  MoveL 10150 to (-40.71, 50.09, 144.49) mm, rotated rx 180 ry 0 rz 180 deg; joints [-39.518, -30.421, 107.234, 74.541, 41.316, -69.786]
  MoveL 10151 to (-40.71, 50.09, 144.49) mm, rotated rx 180 ry 0 rz 180 deg; joints [-39.518, -30.421, 107.234, 74.541, 41.316, -69.786]
  Call Extruder(450.78136)
  MoveL 10152 to (-40.66, 49.79, 144.49) mm, rotated rx -180 ry 0 rz 180 deg; joints [-39.46, -30.443, 107.245, 74.499, 41.265, -69.747]
  MoveL 10153 to (-40.66, 49.79, 144.49) mm, rotated rx -180 ry 0 rz 180 deg; joints [-39.46, -30.443, 107.245, 74.499, 41.265, -69.747]
  Call Extruder(450.94309)
  MoveL 10154 to (-40.61, 49.48, 144.49) mm, rotated rx 180 ry 0 rz 180 deg; joints [-39.402, -30.465, 107.257, 74.456, 41.213, -69.708]
  MoveL 10155 to (-40.61, 49.48, 144.49) mm, rotated rx 180 ry 0 rz 180 deg; joints [-39.402, -30.465, 107.257, 74.456, 41.213, -69.708]
  Call Extruder(451.10554)
  MoveL 10156 to (-40.56, 49.18, 144.49) mm, rotated rx 180 ry 0 rz 180 deg; joints [-39.344, -30.487, 107.268, 74.413, 41.162, -69.669]
  MoveL 10157 to (-40.56, 49.18, 144.49) mm, rotated rx 180 ry 0 rz 180 deg; joints [-39.344, -30.487, 107.268, 74.413, 41.162, -69.669]
  Call Extruder(451.23946)
  MoveL 10158 to (-40.52, 48.93, 144.49) mm, rotated rx 180 ry 0 rz 180 deg; joints [-39.296, -30.504, 107.276, 74.378, 41.118, -69.637]
  MoveL 10159 to (-40.52, 48.93, 144.49) mm, rotated rx 180 ry 0 rz 180 deg; joints [-39.296, -30.504, 107.276, 74.378, 41.118, -69.637]
  Call Extruder(451.37400)
  MoveL 10160 to (-40.47, 48.68, 144.49) mm, rotated rx -180 ry 0 rz 180 deg; joints [-39.247, -30.521, 107.285, 74.343, 41.075, -69.605]
  MoveL 10161 to (-40.47, 48.68, 144.49) mm, rotated rx -180 ry 0 rz 180 deg; joints [-39.247, -30.521, 107.285, 74.343, 41.075, -69.605]
  Call Extruder(451.50914)
  MoveL 10162 to (-40.42, 48.43, 144.49) mm, rotated rx 180 ry 0 rz 180 deg; joints [-39.198, -30.538, 107.293, 74.308, 41.031, -69.574]
  MoveL 10163 to (-40.42, 48.43, 144.49) mm, rotated rx 180 ry 0 rz 180 deg; joints [-39.198, -30.538, 107.293, 74.308, 41.031, -69.574]
  Call Extruder(451.64490)
  MoveL 10164 to (-40.37, 48.18, 144.49) mm, rotated rx 180 ry 0 rz 180 deg; joints [-39.149, -30.555, 107.302, 74.273, 40.988, -69.542]
  MoveL 10165 to (-40.37, 48.18, 144.49) mm, rotated rx 180 ry 0 rz 180 deg; joints [-39.149, -30.555, 107.302, 74.273, 40.988, -69.542]
  Call Extruder(451.78127)
  MoveL 10166 to (-40.32, 47.93, 144.49) mm, rotated rx 180 ry 0 rz 180 deg; joints [-39.1, -30.572, 107.31, 74.237, 40.944, -69.51]
  MoveL 10167 to (-40.32, 47.93, 144.49) mm, rotated rx 180 ry 0 rz 180 deg; joints [-39.1, -30.572, 107.31, 74.237, 40.944, -69.51]
  Call Extruder(451.91824)
  MoveL 10168 to (-40.27, 47.68, 144.49) mm, rotated rx 180 ry 0 rz 180 deg; joints [-39.051, -30.589, 107.319, 74.202, 40.901, -69.478]
  MoveL 10169 to (-40.27, 47.68, 144.49) mm, rotated rx 180 ry 0 rz 180 deg; joints [-39.051, -30.589, 107.319, 74.202, 40.901, -69.478]
  Call Extruder(452.05583)
  MoveL 10170 to (-40.22, 47.43, 144.49) mm, rotated rx -180 ry 0 rz -180 deg; joints [-39.002, -30.605, 107.327, 74.166, 40.857, -69.446]
  MoveL 10171 to (-40.22, 47.43, 144.49) mm, rotated rx -180 ry 0 rz -180 deg; joints [-39.002, -30.605, 107.327, 74.166, 40.857, -69.446]
  Call Extruder(452.16955)
  MoveL 10172 to (-40.17, 47.23, 144.49) mm, rotated rx 180 ry 0 rz 180 deg; joints [-38.962, -30.619, 107.334, 74.137, 40.821, -69.419]
  MoveL 10173 to (-40.17, 47.23, 144.49) mm, rotated rx 180 ry 0 rz 180 deg; joints [-38.962, -30.619, 107.334, 74.137, 40.821, -69.419]
  Call Extruder(452.28373)
  MoveL 10174 to (-40.13, 47.02, 144.49) mm, rotated rx 180 ry 0 rz 180 deg; joints [-38.921, -30.632, 107.341, 74.108, 40.784, -69.393]
  MoveL 10175 to (-40.13, 47.02, 144.49) mm, rotated rx 180 ry 0 rz 180 deg; joints [-38.921, -30.632, 107.341, 74.108, 40.784, -69.393]
  Call Extruder(452.39837)
  MoveL 10176 to (-40.08, 46.82, 144.49) mm, rotated rx -180 ry 0 rz 180 deg; joints [-38.88, -30.645, 107.347, 74.078, 40.748, -69.366]
  MoveL 10177 to (-40.08, 46.82, 144.49) mm, rotated rx -180 ry 0 rz 180 deg; joints [-38.88, -30.645, 107.347, 74.078, 40.748, -69.366]
  Call Extruder(452.51345)
  MoveL 10178 to (-40.04, 46.61, 144.49) mm, rotated rx 180 ry 0 rz 180 deg; joints [-38.839, -30.659, 107.354, 74.049, 40.711, -69.34]
  MoveL 10179 to (-40.04, 46.61, 144.49) mm, rotated rx 180 ry 0 rz 180 deg; joints [-38.839, -30.659, 107.354, 74.049, 40.711, -69.34]
  Call Extruder(452.63569)
  MoveL 10180 to (-39.98, 46.4, 144.49) mm, rotated rx 180 ry 0 rz 180 deg; joints [-38.795, -30.671, 107.36, 74.018, 40.672, -69.312]
  MoveL 10181 to (-39.98, 46.4, 144.49) mm, rotated rx 180 ry 0 rz 180 deg; joints [-38.795, -30.671, 107.36, 74.018, 40.672, -69.312]
  Call Extruder(452.76536)
  MoveL 10182 to (-39.92, 46.18, 144.49) mm, rotated rx 180 ry 0 rz 180 deg; joints [-38.748, -30.684, 107.367, 73.985, 40.629, -69.284]
  MoveL 10183 to (-39.92, 46.18, 144.49) mm, rotated rx 180 ry 0 rz 180 deg; joints [-38.748, -30.684, 107.367, 73.985, 40.629, -69.284]
  Call Extruder(452.89558)
  MoveL 10184 to (-39.85, 45.95, 144.49) mm, rotated rx 180 ry 0 rz 180 deg; joints [-38.7, -30.696, 107.373, 73.953, 40.587, -69.255]
  MoveL 10185 to (-39.85, 45.95, 144.49) mm, rotated rx 180 ry 0 rz 180 deg; joints [-38.7, -30.696, 107.373, 73.953, 40.587, -69.255]
  Call Extruder(453.02638)
  MoveL 10186 to (-39.78, 45.73, 144.49) mm, rotated rx 180 ry 0 rz 180 deg; joints [-38.653, -30.708, 107.379, 73.92, 40.544, -69.226]
  MoveL 10187 to (-39.78, 45.73, 144.49) mm, rotated rx 180 ry 0 rz 180 deg; joints [-38.653, -30.708, 107.379, 73.92, 40.544, -69.226]
  Call Extruder(453.15773)
  MoveL 10188 to (-39.71, 45.51, 144.49) mm, rotated rx 180 ry 0 rz 180 deg; joints [-38.605, -30.721, 107.385, 73.887, 40.501, -69.198]
  MoveL 10189 to (-39.71, 45.51, 144.49) mm, rotated rx 180 ry 0 rz 180 deg; joints [-38.605, -30.721, 107.385, 73.887, 40.501, -69.198]
  Call Extruder(453.26964)
  MoveL 10190 to (-39.65, 45.32, 144.49) mm, rotated rx 180 ry 0 rz 180 deg; joints [-38.565, -30.731, 107.39, 73.859, 40.465, -69.173]
  MoveL 10191 to (-39.65, 45.32, 144.49) mm, rotated rx 180 ry 0 rz 180 deg; joints [-38.565, -30.731, 107.39, 73.859, 40.465, -69.173]
  Call Extruder(453.38198)
  MoveL 10192 to (-39.59, 45.13, 144.49) mm, rotated rx 180 ry 0 rz 180 deg; joints [-38.524, -30.741, 107.395, 73.831, 40.428, -69.149]
  MoveL 10193 to (-39.59, 45.13, 144.49) mm, rotated rx 180 ry 0 rz 180 deg; joints [-38.524, -30.741, 107.395, 73.831, 40.428, -69.149]
  Call Extruder(453.49477)
  MoveL 10194 to (-39.53, 44.94, 144.49) mm, rotated rx -180 ry 0 rz 180 deg; joints [-38.483, -30.75, 107.4, 73.804, 40.391, -69.125]
  MoveL 10195 to (-39.53, 44.94, 144.49) mm, rotated rx -180 ry 0 rz 180 deg; joints [-38.483, -30.75, 107.4, 73.804, 40.391, -69.125]
  Call Extruder(453.60801)
  MoveL 10196 to (-39.47, 44.75, 144.49) mm, rotated rx 180 ry 0 rz 180 deg; joints [-38.443, -30.76, 107.405, 73.776, 40.355, -69.101]
  MoveL 10197 to (-39.47, 44.75, 144.49) mm, rotated rx 180 ry 0 rz 180 deg; joints [-38.443, -30.76, 107.405, 73.776, 40.355, -69.101]
  Call Extruder(453.72169)
  MoveL 10198 to (-39.41, 44.56, 144.49) mm, rotated rx 180 ry 0 rz 180 deg; joints [-38.402, -30.77, 107.41, 73.748, 40.318, -69.076]
  MoveL 10199 to (-39.41, 44.56, 144.49) mm, rotated rx 180 ry 0 rz 180 deg; joints [-38.402, -30.77, 107.41, 73.748, 40.318, -69.076]
  Call Extruder(453.90365)
  MoveL 10200 to (-39.29, 44.27, 144.49) mm, rotated rx 180 ry 0 rz -180 deg; joints [-38.335, -30.782, 107.416, 73.704, 40.258, -69.039]
  MoveL 10201 to (-39.29, 44.27, 144.49) mm, rotated rx 180 ry 0 rz -180 deg; joints [-38.335, -30.782, 107.416, 73.704, 40.258, -69.039]
  Call Extruder(454.08636)
  MoveL 10202 to (-39.17, 43.98, 144.49) mm, rotated rx 180 ry 0 rz 180 deg; joints [-38.269, -30.794, 107.422, 73.66, 40.197, -69.002]
  MoveL 10203 to (-39.17, 43.98, 144.49) mm, rotated rx 180 ry 0 rz 180 deg; joints [-38.269, -30.794, 107.422, 73.66, 40.197, -69.002]
  Call Extruder(454.25678)
  MoveL 10204 to (-39.05, 43.71, 144.49) mm, rotated rx -180 ry 0 rz 180 deg; joints [-38.207, -30.805, 107.427, 73.619, 40.141, -68.967]
  MoveL 10205 to (-39.05, 43.71, 144.49) mm, rotated rx -180 ry 0 rz 180 deg; joints [-38.207, -30.805, 107.427, 73.619, 40.141, -68.967]
  Call Extruder(454.41476)
  MoveL 10206 to (-38.94, 43.46, 144.49) mm, rotated rx 180 ry 0 rz 180 deg; joints [-38.149, -30.815, 107.432, 73.582, 40.089, -68.935]
  MoveL 10207 to (-38.94, 43.46, 144.49) mm, rotated rx 180 ry 0 rz 180 deg; joints [-38.149, -30.815, 107.432, 73.582, 40.089, -68.935]
  Call Extruder(454.57335)
  MoveL 10208 to (-38.84, 43.21, 144.49) mm, rotated rx 180 ry 0 rz 180 deg; joints [-38.092, -30.825, 107.437, 73.544, 40.036, -68.903]
  MoveL 10209 to (-38.84, 43.21, 144.49) mm, rotated rx 180 ry 0 rz 180 deg; joints [-38.092, -30.825, 107.437, 73.544, 40.036, -68.903]
  Call Extruder(454.77952)
  MoveL 10210 to (-38.66, 42.91, 144.49) mm, rotated rx 180 ry 0 rz -180 deg; joints [-38.016, -30.832, 107.441, 73.497, 39.966, -68.865]
  MoveL 10211 to (-38.66, 42.91, 144.49) mm, rotated rx 180 ry 0 rz -180 deg; joints [-38.016, -30.832, 107.441, 73.497, 39.966, -68.865]
  Call Extruder(454.98646)
  MoveL 10212 to (-38.49, 42.6, 144.49) mm, rotated rx 180 ry 0 rz 180 deg; joints [-37.939, -30.839, 107.444, 73.45, 39.896, -68.827]
  MoveL 10213 to (-38.49, 42.6, 144.49) mm, rotated rx 180 ry 0 rz 180 deg; joints [-37.939, -30.839, 107.444, 73.45, 39.896, -68.827]
  Call Extruder(455.19419)
  MoveL 10214 to (-38.31, 42.3, 144.49) mm, rotated rx 180 ry 0 rz 180 deg; joints [-37.863, -30.846, 107.448, 73.403, 39.826, -68.789]
  MoveL 10215 to (-38.31, 42.3, 144.49) mm, rotated rx 180 ry 0 rz 180 deg; joints [-37.863, -30.846, 107.448, 73.403, 39.826, -68.789]
  Call Extruder(455.40269)
  MoveL 10216 to (-38.14, 41.99, 144.49) mm, rotated rx -180 ry 0 rz 180 deg; joints [-37.787, -30.853, 107.451, 73.356, 39.756, -68.751]
  MoveL 10217 to (-38.14, 41.99, 144.49) mm, rotated rx -180 ry 0 rz 180 deg; joints [-37.787, -30.853, 107.451, 73.356, 39.756, -68.751]
  Call Extruder(455.58224)
  MoveL 10218 to (-37.96, 41.75, 144.49) mm, rotated rx 180 ry 0 rz 180 deg; joints [-37.72, -30.854, 107.452, 73.318, 39.694, -68.721]
  MoveL 10219 to (-37.96, 41.75, 144.49) mm, rotated rx 180 ry 0 rz 180 deg; joints [-37.72, -30.854, 107.452, 73.318, 39.694, -68.721]
  Call Extruder(455.91567)
  MoveL 10220 to (-37.63, 41.3, 144.49) mm, rotated rx 180 ry 0 rz 180 deg; joints [-37.598, -30.856, 107.453, 73.247, 39.58, -68.665]
  MoveL 10221 to (-37.63, 41.3, 144.49) mm, rotated rx 180 ry 0 rz 180 deg; joints [-37.598, -30.856, 107.453, 73.247, 39.58, -68.665]
  Call Extruder(456.25030)
  MoveL 10222 to (-37.3, 40.85, 144.49) mm, rotated rx 180 ry 0 rz -180 deg; joints [-37.475, -30.859, 107.454, 73.175, 39.467, -68.61]
  Call Extruder(457.07823)
  MoveL 10223 to (-36.39, 39.81, 144.49) mm, rotated rx 180 ry 0 rz 180 deg; joints [-37.173, -30.845, 107.447, 73.009, 39.183, -68.485]
  Call Extruder(457.90614)
  MoveL 10224 to (-35.35, 38.9, 144.49) mm, rotated rx 180 ry 0 rz 180 deg; joints [-36.876, -30.805, 107.427, 72.859, 38.901, -68.38]
  Call Extruder(458.07344)
  MoveL 10225 to (-35.13, 38.73, 144.49) mm, rotated rx -180 ry 0 rz 180 deg; joints [-36.818, -30.794, 107.422, 72.831, 38.845, -68.363]
  MoveL 10226 to (-35.13, 38.73, 144.49) mm, rotated rx -180 ry 0 rz 180 deg; joints [-36.818, -30.794, 107.422, 72.831, 38.845, -68.363]
  Call Extruder(458.40687)
  MoveL 10227 to (-34.68, 38.4, 144.49) mm, rotated rx 180 ry 0 rz 180 deg; joints [-36.701, -30.77, 107.41, 72.776, 38.733, -68.327]
  MoveL 10228 to (-34.68, 38.4, 144.49) mm, rotated rx 180 ry 0 rz 180 deg; joints [-36.701, -30.77, 107.41, 72.776, 38.733, -68.327]
  Call Extruder(458.73911)
  MoveL 10229 to (-34.22, 38.08, 144.49) mm, rotated rx 180 ry 0 rz 180 deg; joints [-36.584, -30.747, 107.398, 72.721, 38.621, -68.291]
  MoveL 10230 to (-34.22, 38.08, 144.49) mm, rotated rx 180 ry 0 rz 180 deg; joints [-36.584, -30.747, 107.398, 72.721, 38.621, -68.291]
  Call Extruder(458.85681)
  MoveL 10231 to (-34.05, 37.98, 144.49) mm, rotated rx -180 ry 0 rz -180 deg; joints [-36.544, -30.736, 107.393, 72.704, 38.583, -68.281]
  MoveL 10232 to (-34.05, 37.98, 144.49) mm, rotated rx -180 ry 0 rz -180 deg; joints [-36.544, -30.736, 107.393, 72.704, 38.583, -68.281]
  Call Extruder(459.06453)
  MoveL 10233 to (-33.75, 37.8, 144.49) mm, rotated rx -180 ry 0 rz 180 deg; joints [-36.474, -30.716, 107.383, 72.674, 38.514, -68.263]
  MoveL 10234 to (-33.75, 37.8, 144.49) mm, rotated rx -180 ry 0 rz 180 deg; joints [-36.474, -30.716, 107.383, 72.674, 38.514, -68.263]
  Call Extruder(459.27147)
  MoveL 10235 to (-33.45, 37.63, 144.49) mm, rotated rx 180 ry 0 rz 180 deg; joints [-36.403, -30.696, 107.373, 72.644, 38.446, -68.246]
  MoveL 10236 to (-33.45, 37.63, 144.49) mm, rotated rx 180 ry 0 rz 180 deg; joints [-36.403, -30.696, 107.373, 72.644, 38.446, -68.246]
  Call Extruder(459.47764)
  MoveL 10237 to (-33.14, 37.45, 144.49) mm, rotated rx 180 ry 0 rz 180 deg; joints [-36.333, -30.676, 107.363, 72.615, 38.378, -68.228]
  MoveL 10238 to (-33.14, 37.45, 144.49) mm, rotated rx 180 ry 0 rz 180 deg; joints [-36.333, -30.676, 107.363, 72.615, 38.378, -68.228]
  Call Extruder(459.65932)
  MoveL 10239 to (-32.86, 37.31, 144.49) mm, rotated rx 180 ry 0 rz -180 deg; joints [-36.272, -30.656, 107.353, 72.59, 38.318, -68.215]
  MoveL 10240 to (-32.86, 37.31, 144.49) mm, rotated rx 180 ry 0 rz -180 deg; joints [-36.272, -30.656, 107.353, 72.59, 38.318, -68.215]
  Call Extruder(459.81731)
  MoveL 10241 to (-32.62, 37.2, 144.49) mm, rotated rx -180 ry 0 rz 180 deg; joints [-36.221, -30.637, 107.343, 72.571, 38.268, -68.206]
  MoveL 10242 to (-32.62, 37.2, 144.49) mm, rotated rx -180 ry 0 rz 180 deg; joints [-36.221, -30.637, 107.343, 72.571, 38.268, -68.206]
  Call Extruder(459.97470)
  MoveL 10243 to (-32.37, 37.1, 144.49) mm, rotated rx 180 ry 0 rz 180 deg; joints [-36.17, -30.617, 107.333, 72.552, 38.218, -68.197]
  MoveL 10244 to (-32.37, 37.1, 144.49) mm, rotated rx 180 ry 0 rz 180 deg; joints [-36.17, -30.617, 107.333, 72.552, 38.218, -68.197]
  Call Extruder(460.13371)
  MoveL 10245 to (-32.11, 36.99, 144.49) mm, rotated rx 180 ry 0 rz 180 deg; joints [-36.119, -30.597, 107.323, 72.534, 38.167, -68.188]
  MoveL 10246 to (-32.11, 36.99, 144.49) mm, rotated rx 180 ry 0 rz 180 deg; joints [-36.119, -30.597, 107.323, 72.534, 38.167, -68.188]
  Call Extruder(460.28213)
  MoveL 10247 to (-31.87, 36.89, 144.49) mm, rotated rx 180 ry 0 rz -180 deg; joints [-36.071, -30.578, 107.313, 72.517, 38.12, -68.18]
  MoveL 10248 to (-31.87, 36.89, 144.49) mm, rotated rx 180 ry 0 rz -180 deg; joints [-36.071, -30.578, 107.313, 72.517, 38.12, -68.18]
  Call Extruder(460.43006)
  MoveL 10249 to (-31.64, 36.79, 144.49) mm, rotated rx 180 ry 0 rz 180 deg; joints [-36.023, -30.559, 107.304, 72.499, 38.073, -68.172]
  MoveL 10250 to (-31.64, 36.79, 144.49) mm, rotated rx 180 ry 0 rz 180 deg; joints [-36.023, -30.559, 107.304, 72.499, 38.073, -68.172]
  Call Extruder(460.54351)
  MoveL 10251 to (-31.45, 36.73, 144.49) mm, rotated rx 180 ry 0 rz 180 deg; joints [-35.989, -30.542, 107.296, 72.488, 38.038, -68.168]
  MoveL 10252 to (-31.45, 36.73, 144.49) mm, rotated rx 180 ry 0 rz 180 deg; joints [-35.989, -30.542, 107.296, 72.488, 38.038, -68.168]
  Call Extruder(460.65653)
  MoveL 10253 to (-31.26, 36.67, 144.49) mm, rotated rx 180 ry 0 rz 180 deg; joints [-35.954, -30.526, 107.287, 72.477, 38.003, -68.165]
  MoveL 10254 to (-31.26, 36.67, 144.49) mm, rotated rx 180 ry 0 rz 180 deg; joints [-35.954, -30.526, 107.287, 72.477, 38.003, -68.165]
  Call Extruder(460.76910)
  MoveL 10255 to (-31.07, 36.61, 144.49) mm, rotated rx 180 ry 0 rz 180 deg; joints [-35.919, -30.509, 107.279, 72.466, 37.968, -68.161]
  MoveL 10256 to (-31.07, 36.61, 144.49) mm, rotated rx 180 ry 0 rz 180 deg; joints [-35.919, -30.509, 107.279, 72.466, 37.968, -68.161]
  Call Extruder(460.88122)
  MoveL 10257 to (-30.88, 36.55, 144.49) mm, rotated rx 180 ry 0 rz 180 deg; joints [-35.884, -30.493, 107.27, 72.455, 37.933, -68.157]
  MoveL 10258 to (-30.88, 36.55, 144.49) mm, rotated rx 180 ry 0 rz 180 deg; joints [-35.884, -30.493, 107.27, 72.455, 37.933, -68.157]
  Call Extruder(460.99290)
  MoveL 10259 to (-30.7, 36.49, 144.49) mm, rotated rx -180 ry 0 rz 180 deg; joints [-35.849, -30.476, 107.262, 72.444, 37.898, -68.153]
  MoveL 10260 to (-30.7, 36.49, 144.49) mm, rotated rx -180 ry 0 rz 180 deg; joints [-35.849, -30.476, 107.262, 72.444, 37.898, -68.153]
  Call Extruder(461.12397)
  MoveL 10261 to (-30.47, 36.42, 144.49) mm, rotated rx -180 ry 0 rz 180 deg; joints [-35.809, -30.456, 107.252, 72.432, 37.858, -68.149]
  MoveL 10262 to (-30.47, 36.42, 144.49) mm, rotated rx -180 ry 0 rz 180 deg; joints [-35.809, -30.456, 107.252, 72.432, 37.858, -68.149]
  Call Extruder(461.25448)
  MoveL 10263 to (-30.25, 36.35, 144.49) mm, rotated rx -180 ry 0 rz 180 deg; joints [-35.768, -30.436, 107.242, 72.42, 37.818, -68.145]
  MoveL 10264 to (-30.25, 36.35, 144.49) mm, rotated rx -180 ry 0 rz 180 deg; joints [-35.768, -30.436, 107.242, 72.42, 37.818, -68.145]
  Call Extruder(461.38443)
  MoveL 10265 to (-30.02, 36.28, 144.49) mm, rotated rx -180 ry 0 rz 180 deg; joints [-35.728, -30.416, 107.232, 72.407, 37.777, -68.141]
  MoveL 10266 to (-30.02, 36.28, 144.49) mm, rotated rx -180 ry 0 rz 180 deg; joints [-35.728, -30.416, 107.232, 72.407, 37.777, -68.141]
  Call Extruder(461.51381)
  MoveL 10267 to (-29.8, 36.22, 144.49) mm, rotated rx 180 ry 0 rz 180 deg; joints [-35.688, -30.395, 107.221, 72.395, 37.737, -68.137]
  MoveL 10268 to (-29.8, 36.22, 144.49) mm, rotated rx 180 ry 0 rz 180 deg; joints [-35.688, -30.395, 107.221, 72.395, 37.737, -68.137]
  Call Extruder(461.63577)
  MoveL 10269 to (-29.59, 36.16, 144.49) mm, rotated rx 180 ry 0 rz 180 deg; joints [-35.651, -30.375, 107.211, 72.385, 37.699, -68.135]
  MoveL 10270 to (-29.59, 36.16, 144.49) mm, rotated rx 180 ry 0 rz 180 deg; joints [-35.651, -30.375, 107.211, 72.385, 37.699, -68.135]
  Call Extruder(461.75062)
  MoveL 10271 to (-29.38, 36.12, 144.49) mm, rotated rx 180 ry 0 rz 180 deg; joints [-35.617, -30.356, 107.201, 72.377, 37.665, -68.134]
  MoveL 10272 to (-29.38, 36.12, 144.49) mm, rotated rx 180 ry 0 rz 180 deg; joints [-35.617, -30.356, 107.201, 72.377, 37.665, -68.134]
  Call Extruder(461.86501)
  MoveL 10273 to (-29.18, 36.07, 144.49) mm, rotated rx 180 ry 0 rz 180 deg; joints [-35.584, -30.336, 107.191, 72.368, 37.631, -68.133]
  MoveL 10274 to (-29.18, 36.07, 144.49) mm, rotated rx 180 ry 0 rz 180 deg; joints [-35.584, -30.336, 107.191, 72.368, 37.631, -68.133]
  Call Extruder(461.97895)
  MoveL 10275 to (-28.97, 36.03, 144.49) mm, rotated rx 180 ry 0 rz 180 deg; joints [-35.55, -30.316, 107.181, 72.36, 37.597, -68.132]
  MoveL 10276 to (-28.97, 36.03, 144.49) mm, rotated rx 180 ry 0 rz 180 deg; joints [-35.55, -30.316, 107.181, 72.36, 37.597, -68.132]
  Call Extruder(462.09244)
  MoveL 10277 to (-28.77, 35.98, 144.49) mm, rotated rx 180 ry 0 rz 180 deg; joints [-35.517, -30.296, 107.171, 72.351, 37.563, -68.131]
  MoveL 10278 to (-28.77, 35.98, 144.49) mm, rotated rx 180 ry 0 rz 180 deg; joints [-35.517, -30.296, 107.171, 72.351, 37.563, -68.131]
  Call Extruder(462.22973)
  MoveL 10279 to (-28.52, 35.93, 144.49) mm, rotated rx 180 ry 0 rz 180 deg; joints [-35.477, -30.271, 107.158, 72.342, 37.522, -68.131]
  MoveL 10280 to (-28.52, 35.93, 144.49) mm, rotated rx 180 ry 0 rz 180 deg; joints [-35.477, -30.271, 107.158, 72.342, 37.522, -68.131]
  Call Extruder(462.36640)
  MoveL 10281 to (-28.27, 35.88, 144.49) mm, rotated rx 180 ry 0 rz -180 deg; joints [-35.437, -30.246, 107.146, 72.333, 37.481, -68.131]
  MoveL 10282 to (-28.27, 35.88, 144.49) mm, rotated rx 180 ry 0 rz -180 deg; joints [-35.437, -30.246, 107.146, 72.333, 37.481, -68.131]
  Call Extruder(462.50246)
  MoveL 10283 to (-28.02, 35.83, 144.49) mm, rotated rx 180 ry 0 rz 180 deg; joints [-35.397, -30.222, 107.133, 72.323, 37.441, -68.13]
  MoveL 10284 to (-28.02, 35.83, 144.49) mm, rotated rx 180 ry 0 rz 180 deg; joints [-35.397, -30.222, 107.133, 72.323, 37.441, -68.13]
  Call Extruder(462.63791)
  MoveL 10285 to (-27.77, 35.78, 144.49) mm, rotated rx 180 ry 0 rz 180 deg; joints [-35.357, -30.197, 107.121, 72.314, 37.4, -68.13]
  MoveL 10286 to (-27.77, 35.78, 144.49) mm, rotated rx 180 ry 0 rz 180 deg; joints [-35.357, -30.197, 107.121, 72.314, 37.4, -68.13]
  Call Extruder(462.77275)
  MoveL 10287 to (-27.52, 35.73, 144.49) mm, rotated rx 180 ry 0 rz 180 deg; joints [-35.317, -30.172, 107.108, 72.305, 37.359, -68.13]
  MoveL 10288 to (-27.52, 35.73, 144.49) mm, rotated rx 180 ry 0 rz 180 deg; joints [-35.317, -30.172, 107.108, 72.305, 37.359, -68.13]
  Call Extruder(462.90698)
  MoveL 10289 to (-27.27, 35.68, 144.49) mm, rotated rx 180 ry 0 rz 180 deg; joints [-35.277, -30.147, 107.095, 72.296, 37.319, -68.129]
  MoveL 10290 to (-27.27, 35.68, 144.49) mm, rotated rx 180 ry 0 rz 180 deg; joints [-35.277, -30.147, 107.095, 72.296, 37.319, -68.129]
  Call Extruder(463.04061)
  MoveL 10291 to (-27.03, 35.64, 144.49) mm, rotated rx 180 ry 0 rz 180 deg; joints [-35.238, -30.123, 107.083, 72.286, 37.278, -68.129]
  MoveL 10292 to (-27.03, 35.64, 144.49) mm, rotated rx 180 ry 0 rz 180 deg; joints [-35.238, -30.123, 107.083, 72.286, 37.278, -68.129]
  Call Extruder(463.20270)
  MoveL 10293 to (-26.72, 35.59, 144.49) mm, rotated rx 180 ry 0 rz 180 deg; joints [-35.191, -30.091, 107.067, 72.277, 37.23, -68.13]
  MoveL 10294 to (-26.72, 35.59, 144.49) mm, rotated rx 180 ry 0 rz 180 deg; joints [-35.191, -30.091, 107.067, 72.277, 37.23, -68.13]
  Call Extruder(463.36408)
  MoveL 10295 to (-26.41, 35.54, 144.49) mm, rotated rx 180 ry 0 rz 180 deg; joints [-35.145, -30.059, 107.05, 72.268, 37.183, -68.132]
  MoveL 10296 to (-26.41, 35.54, 144.49) mm, rotated rx 180 ry 0 rz 180 deg; joints [-35.145, -30.059, 107.05, 72.268, 37.183, -68.132]
  Call Extruder(463.52472)
  MoveL 10297 to (-26.11, 35.49, 144.49) mm, rotated rx 180 ry 0 rz -180 deg; joints [-35.098, -30.028, 107.034, 72.259, 37.135, -68.134]
  MoveL 10298 to (-26.11, 35.49, 144.49) mm, rotated rx 180 ry 0 rz -180 deg; joints [-35.098, -30.028, 107.034, 72.259, 37.135, -68.134]
  Call Extruder(463.68463)
  MoveL 10299 to (-25.8, 35.44, 144.49) mm, rotated rx 180 ry 0 rz 180 deg; joints [-35.052, -29.996, 107.018, 72.25, 37.087, -68.135]
  MoveL 10300 to (-25.8, 35.44, 144.49) mm, rotated rx 180 ry 0 rz 180 deg; joints [-35.052, -29.996, 107.018, 72.25, 37.087, -68.135]
  Call Extruder(463.84382)
  MoveL 10301 to (-25.5, 35.39, 144.49) mm, rotated rx 180 ry 0 rz 180 deg; joints [-35.006, -29.965, 107.002, 72.24, 37.04, -68.137]
  MoveL 10302 to (-25.5, 35.39, 144.49) mm, rotated rx 180 ry 0 rz 180 deg; joints [-35.006, -29.965, 107.002, 72.24, 37.04, -68.137]
  Call Extruder(464.00228)
  MoveL 10303 to (-25.19, 35.34, 144.49) mm, rotated rx 180 ry 0 rz 180 deg; joints [-34.96, -29.933, 106.986, 72.231, 36.992, -68.138]
  MoveL 10304 to (-25.19, 35.34, 144.49) mm, rotated rx 180 ry 0 rz 180 deg; joints [-34.96, -29.933, 106.986, 72.231, 36.992, -68.138]
  Call Extruder(464.20116)
  MoveL 10305 to (-24.8, 35.3, 144.49) mm, rotated rx 180 ry 0 rz 180 deg; joints [-34.904, -29.892, 106.964, 72.222, 36.935, -68.143]
  MoveL 10306 to (-24.8, 35.3, 144.49) mm, rotated rx 180 ry 0 rz 180 deg; joints [-34.904, -29.892, 106.964, 72.222, 36.935, -68.143]
  Call Extruder(464.39916)
  MoveL 10307 to (-24.42, 35.25, 144.49) mm, rotated rx 180 ry 0 rz 180 deg; joints [-34.849, -29.85, 106.943, 72.214, 36.877, -68.147]
  MoveL 10308 to (-24.42, 35.25, 144.49) mm, rotated rx 180 ry 0 rz 180 deg; joints [-34.849, -29.85, 106.943, 72.214, 36.877, -68.147]
  Call Extruder(464.59630)
  MoveL 10309 to (-24.03, 35.21, 144.49) mm, rotated rx 180 ry 0 rz 180 deg; joints [-34.794, -29.809, 106.922, 72.205, 36.819, -68.152]
  MoveL 10310 to (-24.03, 35.21, 144.49) mm, rotated rx 180 ry 0 rz 180 deg; joints [-34.794, -29.809, 106.922, 72.205, 36.819, -68.152]
  Call Extruder(464.79258)
  MoveL 10311 to (-23.64, 35.16, 144.49) mm, rotated rx -180 ry 0 rz 180 deg; joints [-34.738, -29.767, 106.9, 72.196, 36.762, -68.156]
  MoveL 10312 to (-23.64, 35.16, 144.49) mm, rotated rx -180 ry 0 rz 180 deg; joints [-34.738, -29.767, 106.9, 72.196, 36.762, -68.156]
  Call Extruder(465.03826)
  MoveL 10313 to (-23.15, 35.11, 144.49) mm, rotated rx -180 ry 0 rz 180 deg; joints [-34.671, -29.714, 106.873, 72.187, 36.692, -68.163]
  MoveL 10314 to (-23.15, 35.11, 144.49) mm, rotated rx -180 ry 0 rz 180 deg; joints [-34.671, -29.714, 106.873, 72.187, 36.692, -68.163]
  Call Extruder(465.33299)
  MoveL 10315 to (-22.56, 35.07, 144.49) mm, rotated rx 180 ry 0 rz 180 deg; joints [-34.592, -29.649, 106.839, 72.178, 36.608, -68.174]
  MoveL 10316 to (-22.56, 35.07, 144.49) mm, rotated rx 180 ry 0 rz 180 deg; joints [-34.592, -29.649, 106.839, 72.178, 36.608, -68.174]
  Call Extruder(465.62639)
  MoveL 10317 to (-21.97, 35.02, 144.49) mm, rotated rx 180 ry 0 rz -180 deg; joints [-34.512, -29.583, 106.805, 72.169, 36.525, -68.184]
  MoveL 10318 to (-21.97, 35.02, 144.49) mm, rotated rx 180 ry 0 rz -180 deg; joints [-34.512, -29.583, 106.805, 72.169, 36.525, -68.184]
  Call Extruder(466.05972)
  MoveL 10319 to (-21.1, 34.97, 144.49) mm, rotated rx -180 ry 0 rz 180 deg; joints [-34.399, -29.484, 106.753, 72.159, 36.406, -68.204]
  MoveL 10320 to (-21.1, 34.97, 144.49) mm, rotated rx -180 ry 0 rz 180 deg; joints [-34.399, -29.484, 106.753, 72.159, 36.406, -68.204]
  Call Extruder(466.63188)
  MoveL 10321 to (-19.94, 34.93, 144.49) mm, rotated rx -180 ry 0 rz 180 deg; joints [-34.253, -29.351, 106.684, 72.15, 36.25, -68.232]
  MoveL 10322 to (-19.94, 34.93, 144.49) mm, rotated rx -180 ry 0 rz 180 deg; joints [-34.253, -29.351, 106.684, 72.15, 36.25, -68.232]
  Call Extruder(467.05971)
  MoveL 10323 to (-19.06, 34.91, 144.49) mm, rotated rx -180 ry 0 rz 180 deg; joints [-34.146, -29.25, 106.631, 72.146, 36.136, -68.256]
  Call Extruder(583.70842)
  MoveL 10324 to (219.06, 34.91, 144.49) mm, rotated rx -180 ry 0 rz 180 deg; joints [-18.248, 2.992, 81.238, 73.041, 19.109, -72.114]
  MoveL 10325 to (219.06, 34.91, 144.49) mm, rotated rx -180 ry 0 rz 180 deg; joints [-18.248, 2.992, 81.238, 73.041, 19.109, -72.114]
  Call Extruder(584.42399)
  MoveL 10326 to (220.52, 34.95, 144.49) mm, rotated rx 180 ry 0 rz 180 deg; joints [-18.199, 3.215, 81.003, 72.964, 19.066, -72.038]
  MoveL 10327 to (220.52, 34.95, 144.49) mm, rotated rx 180 ry 0 rz 180 deg; joints [-18.199, 3.215, 81.003, 72.964, 19.066, -72.038]
  Call Extruder(584.99873)
  MoveL 10328 to (221.68, 35, 144.49) mm, rotated rx 180 ry 0 rz -180 deg; joints [-18.162, 3.394, 80.815, 72.903, 19.033, -71.976]
  MoveL 10329 to (221.68, 35, 144.49) mm, rotated rx 180 ry 0 rz -180 deg; joints [-18.162, 3.394, 80.815, 72.903, 19.033, -71.976]
  Call Extruder(585.29212)
  MoveL 10330 to (222.27, 35.04, 144.49) mm, rotated rx 180 ry 0 rz 180 deg; joints [-18.146, 3.486, 80.717, 72.873, 19.019, -71.947]
  MoveL 10331 to (222.27, 35.04, 144.49) mm, rotated rx 180 ry 0 rz 180 deg; joints [-18.146, 3.486, 80.717, 72.873, 19.019, -71.947]
  Call Extruder(585.58685)
  MoveL 10332 to (222.86, 35.09, 144.49) mm, rotated rx 180 ry 0 rz 180 deg; joints [-18.13, 3.579, 80.62, 72.843, 19.006, -71.916]
  MoveL 10333 to (222.86, 35.09, 144.49) mm, rotated rx 180 ry 0 rz 180 deg; joints [-18.13, 3.579, 80.62, 72.843, 19.006, -71.916]
  Call Extruder(585.88292)
  MoveL 10334 to (223.45, 35.14, 144.49) mm, rotated rx 180 ry 0 rz 180 deg; joints [-18.113, 3.671, 80.522, 72.812, 18.992, -71.886]
  MoveL 10335 to (223.45, 35.14, 144.49) mm, rotated rx 180 ry 0 rz 180 deg; joints [-18.113, 3.671, 80.522, 72.812, 18.992, -71.886]
  Call Extruder(586.07919)
  MoveL 10336 to (223.84, 35.18, 144.49) mm, rotated rx 180 ry 0 rz 180 deg; joints [-18.104, 3.732, 80.457, 72.794, 18.984, -71.867]
  MoveL 10337 to (223.84, 35.18, 144.49) mm, rotated rx 180 ry 0 rz 180 deg; joints [-18.104, 3.732, 80.457, 72.794, 18.984, -71.867]
  Call Extruder(586.27633)
  MoveL 10338 to (224.22, 35.23, 144.49) mm, rotated rx 180 ry 0 rz 180 deg; joints [-18.095, 3.794, 80.391, 72.775, 18.977, -71.848]
  MoveL 10339 to (224.22, 35.23, 144.49) mm, rotated rx 180 ry 0 rz 180 deg; joints [-18.095, 3.794, 80.391, 72.775, 18.977, -71.848]
  Call Extruder(586.47434)
  MoveL 10340 to (224.61, 35.27, 144.49) mm, rotated rx -180 ry 0 rz 180 deg; joints [-18.087, 3.855, 80.326, 72.756, 18.97, -71.829]
  MoveL 10341 to (224.61, 35.27, 144.49) mm, rotated rx -180 ry 0 rz 180 deg; joints [-18.087, 3.855, 80.326, 72.756, 18.97, -71.829]
  Call Extruder(586.67322)
  MoveL 10342 to (225, 35.32, 144.49) mm, rotated rx 180 ry 0 rz 180 deg; joints [-18.078, 3.917, 80.261, 72.736, 18.962, -71.809]
  MoveL 10343 to (225, 35.32, 144.49) mm, rotated rx 180 ry 0 rz 180 deg; joints [-18.078, 3.917, 80.261, 72.736, 18.962, -71.809]
  Call Extruder(586.85230)
  MoveL 10344 to (225.34, 35.37, 144.49) mm, rotated rx 180 ry 0 rz 180 deg; joints [-18.07, 3.972, 80.202, 72.719, 18.956, -71.792]
  MoveL 10345 to (225.34, 35.37, 144.49) mm, rotated rx 180 ry 0 rz 180 deg; joints [-18.07, 3.972, 80.202, 72.719, 18.956, -71.792]
  Call Extruder(587.01148)
  MoveL 10346 to (225.65, 35.42, 144.49) mm, rotated rx 180 ry 0 rz 180 deg; joints [-18.065, 4.022, 80.149, 72.705, 18.952, -71.778]
  MoveL 10347 to (225.65, 35.42, 144.49) mm, rotated rx 180 ry 0 rz 180 deg; joints [-18.065, 4.022, 80.149, 72.705, 18.952, -71.778]
  Call Extruder(587.17139)
  MoveL 10348 to (225.96, 35.46, 144.49) mm, rotated rx -180 ry 0 rz 180 deg; joints [-18.059, 4.071, 80.097, 72.691, 18.948, -71.763]
  MoveL 10349 to (225.96, 35.46, 144.49) mm, rotated rx -180 ry 0 rz 180 deg; joints [-18.059, 4.071, 80.097, 72.691, 18.948, -71.763]
  Call Extruder(587.33203)
  MoveL 10350 to (226.26, 35.51, 144.49) mm, rotated rx -180 ry 0 rz 180 deg; joints [-18.054, 4.12, 80.044, 72.676, 18.943, -71.749]
  MoveL 10351 to (226.26, 35.51, 144.49) mm, rotated rx -180 ry 0 rz 180 deg; joints [-18.054, 4.12, 80.044, 72.676, 18.943, -71.749]
  Call Extruder(587.49340)
  MoveL 10352 to (226.57, 35.56, 144.49) mm, rotated rx 180 ry 0 rz 180 deg; joints [-18.048, 4.17, 79.992, 72.662, 18.939, -71.734]
  MoveL 10353 to (226.57, 35.56, 144.49) mm, rotated rx 180 ry 0 rz 180 deg; joints [-18.048, 4.17, 79.992, 72.662, 18.939, -71.734]
  Call Extruder(587.65549)
  MoveL 10354 to (226.87, 35.61, 144.49) mm, rotated rx 180 ry 0 rz -180 deg; joints [-18.042, 4.219, 79.939, 72.647, 18.935, -71.719]
  MoveL 10355 to (226.87, 35.61, 144.49) mm, rotated rx 180 ry 0 rz -180 deg; joints [-18.042, 4.219, 79.939, 72.647, 18.935, -71.719]
  Call Extruder(587.80369)
  MoveL 10356 to (227.15, 35.66, 144.49) mm, rotated rx 180 ry 0 rz 180 deg; joints [-18.038, 4.264, 79.891, 72.634, 18.931, -71.705]
  MoveL 10357 to (227.15, 35.66, 144.49) mm, rotated rx 180 ry 0 rz 180 deg; joints [-18.038, 4.264, 79.891, 72.634, 18.931, -71.705]
  Call Extruder(587.93792)
  MoveL 10358 to (227.4, 35.71, 144.49) mm, rotated rx 180 ry 0 rz 180 deg; joints [-18.034, 4.305, 79.847, 72.623, 18.929, -71.694]
  MoveL 10359 to (227.4, 35.71, 144.49) mm, rotated rx 180 ry 0 rz 180 deg; joints [-18.034, 4.305, 79.847, 72.623, 18.929, -71.694]
  Call Extruder(588.07276)
  MoveL 10360 to (227.65, 35.76, 144.49) mm, rotated rx 180 ry 0 rz 180 deg; joints [-18.031, 4.345, 79.804, 72.612, 18.926, -71.682]
  MoveL 10361 to (227.65, 35.76, 144.49) mm, rotated rx 180 ry 0 rz 180 deg; joints [-18.031, 4.345, 79.804, 72.612, 18.926, -71.682]
  Call Extruder(588.20822)
  MoveL 10362 to (227.9, 35.81, 144.49) mm, rotated rx 180 ry 0 rz -180 deg; joints [-18.027, 4.386, 79.76, 72.6, 18.924, -71.671]
  MoveL 10363 to (227.9, 35.81, 144.49) mm, rotated rx 180 ry 0 rz -180 deg; joints [-18.027, 4.386, 79.76, 72.6, 18.924, -71.671]
  Call Extruder(588.34428)
  MoveL 10364 to (228.15, 35.86, 144.49) mm, rotated rx -180 ry 0 rz 180 deg; joints [-18.024, 4.427, 79.717, 72.589, 18.921, -71.659]
  MoveL 10365 to (228.15, 35.86, 144.49) mm, rotated rx -180 ry 0 rz 180 deg; joints [-18.024, 4.427, 79.717, 72.589, 18.921, -71.659]
  Call Extruder(588.48095)
  MoveL 10366 to (228.4, 35.91, 144.49) mm, rotated rx 180 ry 0 rz 180 deg; joints [-18.02, 4.468, 79.673, 72.577, 18.919, -71.647]
  MoveL 10367 to (228.4, 35.91, 144.49) mm, rotated rx 180 ry 0 rz 180 deg; joints [-18.02, 4.468, 79.673, 72.577, 18.919, -71.647]
  Call Extruder(588.61823)
  MoveL 10368 to (228.64, 35.96, 144.49) mm, rotated rx 180 ry 0 rz -180 deg; joints [-18.017, 4.508, 79.629, 72.566, 18.917, -71.635]
  MoveL 10369 to (228.64, 35.96, 144.49) mm, rotated rx 180 ry 0 rz -180 deg; joints [-18.017, 4.508, 79.629, 72.566, 18.917, -71.635]
  Call Extruder(588.74391)
  MoveL 10370 to (228.87, 36, 144.49) mm, rotated rx 180 ry 0 rz 180 deg; joints [-18.014, 4.546, 79.589, 72.555, 18.915, -71.625]
  MoveL 10371 to (228.87, 36, 144.49) mm, rotated rx 180 ry 0 rz 180 deg; joints [-18.014, 4.546, 79.589, 72.555, 18.915, -71.625]
  Call Extruder(588.85785)
  MoveL 10372 to (229.08, 36.05, 144.49) mm, rotated rx 180 ry 0 rz -180 deg; joints [-18.012, 4.579, 79.553, 72.546, 18.913, -71.615]
  MoveL 10373 to (229.08, 36.05, 144.49) mm, rotated rx 180 ry 0 rz -180 deg; joints [-18.012, 4.579, 79.553, 72.546, 18.913, -71.615]
  Call Extruder(588.97225)
  MoveL 10374 to (229.28, 36.09, 144.49) mm, rotated rx 180 ry 0 rz 180 deg; joints [-18.009, 4.613, 79.517, 72.537, 18.912, -71.606]
  MoveL 10375 to (229.28, 36.09, 144.49) mm, rotated rx 180 ry 0 rz 180 deg; joints [-18.009, 4.613, 79.517, 72.537, 18.912, -71.606]
  Call Extruder(589.08710)
  MoveL 10376 to (229.48, 36.14, 144.49) mm, rotated rx -180 ry 0 rz 180 deg; joints [-18.007, 4.647, 79.481, 72.527, 18.91, -71.596]
  MoveL 10377 to (229.48, 36.14, 144.49) mm, rotated rx -180 ry 0 rz 180 deg; joints [-18.007, 4.647, 79.481, 72.527, 18.91, -71.596]
  Call Extruder(589.20240)
  MoveL 10378 to (229.69, 36.18, 144.49) mm, rotated rx -180 ry 0 rz 180 deg; joints [-18.005, 4.68, 79.445, 72.518, 18.909, -71.586]
  MoveL 10379 to (229.69, 36.18, 144.49) mm, rotated rx -180 ry 0 rz 180 deg; joints [-18.005, 4.68, 79.445, 72.518, 18.909, -71.586]
  Call Extruder(589.26695)
  MoveL 10380 to (229.8, 36.22, 144.49) mm, rotated rx 180 ry 0 rz 180 deg; joints [-18.004, 4.699, 79.424, 72.514, 18.909, -71.582]
  MoveL 10381 to (229.8, 36.22, 144.49) mm, rotated rx 180 ry 0 rz 180 deg; joints [-18.004, 4.699, 79.424, 72.514, 18.909, -71.582]
  Call Extruder(589.39662)
  MoveL 10382 to (230.02, 36.28, 144.49) mm, rotated rx -180 ry 0 rz -180 deg; joints [-18.004, 4.737, 79.383, 72.505, 18.909, -71.573]
  MoveL 10383 to (230.02, 36.28, 144.49) mm, rotated rx -180 ry 0 rz -180 deg; joints [-18.004, 4.737, 79.383, 72.505, 18.909, -71.573]
  Call Extruder(589.52685)
  MoveL 10384 to (230.25, 36.35, 144.49) mm, rotated rx 180 ry 0 rz 180 deg; joints [-18.003, 4.775, 79.343, 72.497, 18.91, -71.564]
  MoveL 10385 to (230.25, 36.35, 144.49) mm, rotated rx 180 ry 0 rz 180 deg; joints [-18.003, 4.775, 79.343, 72.497, 18.91, -71.564]
  Call Extruder(589.65764)
  MoveL 10386 to (230.47, 36.42, 144.49) mm, rotated rx 180 ry 0 rz 180 deg; joints [-18.003, 4.813, 79.302, 72.488, 18.91, -71.555]
  MoveL 10387 to (230.47, 36.42, 144.49) mm, rotated rx 180 ry 0 rz 180 deg; joints [-18.003, 4.813, 79.302, 72.488, 18.91, -71.555]
  Call Extruder(589.78900)
  MoveL 10388 to (230.7, 36.49, 144.49) mm, rotated rx -180 ry 0 rz 180 deg; joints [-18.002, 4.851, 79.261, 72.479, 18.91, -71.545]
  MoveL 10389 to (230.7, 36.49, 144.49) mm, rotated rx -180 ry 0 rz 180 deg; joints [-18.002, 4.851, 79.261, 72.479, 18.91, -71.545]
  Call Extruder(589.90090)
  MoveL 10390 to (230.88, 36.55, 144.49) mm, rotated rx 180 ry 0 rz 180 deg; joints [-18.002, 4.883, 79.226, 72.472, 18.911, -71.538]
  MoveL 10391 to (230.88, 36.55, 144.49) mm, rotated rx 180 ry 0 rz 180 deg; joints [-18.002, 4.883, 79.226, 72.472, 18.911, -71.538]
  Call Extruder(590.01324)
  MoveL 10392 to (231.07, 36.61, 144.49) mm, rotated rx 180 ry 0 rz 180 deg; joints [-18.002, 4.915, 79.192, 72.465, 18.912, -71.53]
  MoveL 10393 to (231.07, 36.61, 144.49) mm, rotated rx 180 ry 0 rz 180 deg; joints [-18.002, 4.915, 79.192, 72.465, 18.912, -71.53]
  Call Extruder(590.12603)
  MoveL 10394 to (231.26, 36.67, 144.49) mm, rotated rx -180 ry 0 rz 180 deg; joints [-18.002, 4.947, 79.157, 72.458, 18.913, -71.523]
  MoveL 10395 to (231.26, 36.67, 144.49) mm, rotated rx -180 ry 0 rz 180 deg; joints [-18.002, 4.947, 79.157, 72.458, 18.913, -71.523]
  Call Extruder(590.23926)
  MoveL 10396 to (231.45, 36.73, 144.49) mm, rotated rx 180 ry 0 rz 180 deg; joints [-18.002, 4.979, 79.122, 72.451, 18.913, -71.515]
  MoveL 10397 to (231.45, 36.73, 144.49) mm, rotated rx 180 ry 0 rz 180 deg; joints [-18.002, 4.979, 79.122, 72.451, 18.913, -71.515]
  Call Extruder(590.35294)
  MoveL 10398 to (231.64, 36.79, 144.49) mm, rotated rx -180 ry 0 rz 180 deg; joints [-18.002, 5.011, 79.088, 72.443, 18.914, -71.508]
  MoveL 10399 to (231.64, 36.79, 144.49) mm, rotated rx -180 ry 0 rz 180 deg; joints [-18.002, 5.011, 79.088, 72.443, 18.914, -71.508]
  Call Extruder(590.53490)
  MoveL 10400 to (231.93, 36.91, 144.49) mm, rotated rx -180 ry 0 rz 180 deg; joints [-18.005, 5.062, 79.032, 72.435, 18.918, -71.498]
  MoveL 10401 to (231.93, 36.91, 144.49) mm, rotated rx -180 ry 0 rz 180 deg; joints [-18.005, 5.062, 79.032, 72.435, 18.918, -71.498]
  Call Extruder(590.71761)
  MoveL 10402 to (232.22, 37.04, 144.49) mm, rotated rx 180 ry 0 rz 180 deg; joints [-18.008, 5.114, 78.977, 72.426, 18.922, -71.488]
  MoveL 10403 to (232.22, 37.04, 144.49) mm, rotated rx 180 ry 0 rz 180 deg; joints [-18.008, 5.114, 78.977, 72.426, 18.922, -71.488]
  Call Extruder(590.88803)
  MoveL 10404 to (232.49, 37.15, 144.49) mm, rotated rx 180 ry 0 rz 180 deg; joints [-18.011, 5.161, 78.925, 72.417, 18.926, -71.479]
  MoveL 10405 to (232.49, 37.15, 144.49) mm, rotated rx 180 ry 0 rz 180 deg; joints [-18.011, 5.161, 78.925, 72.417, 18.926, -71.479]
  Call Extruder(591.04603)
  MoveL 10406 to (232.74, 37.26, 144.49) mm, rotated rx 180 ry 0 rz -180 deg; joints [-18.013, 5.205, 78.878, 72.41, 18.93, -71.471]
  MoveL 10407 to (232.74, 37.26, 144.49) mm, rotated rx 180 ry 0 rz -180 deg; joints [-18.013, 5.205, 78.878, 72.41, 18.93, -71.471]
  Call Extruder(591.20464)
  MoveL 10408 to (232.99, 37.36, 144.49) mm, rotated rx -180 ry 0 rz 180 deg; joints [-18.016, 5.249, 78.83, 72.402, 18.933, -71.463]
  MoveL 10409 to (232.99, 37.36, 144.49) mm, rotated rx -180 ry 0 rz 180 deg; joints [-18.016, 5.249, 78.83, 72.402, 18.933, -71.463]
  Call Extruder(591.41080)
  MoveL 10410 to (233.29, 37.54, 144.49) mm, rotated rx 180 ry 0 rz -180 deg; joints [-18.024, 5.305, 78.77, 72.397, 18.943, -71.457]
  MoveL 10411 to (233.29, 37.54, 144.49) mm, rotated rx 180 ry 0 rz -180 deg; joints [-18.024, 5.305, 78.77, 72.397, 18.943, -71.457]
  Call Extruder(591.61775)
  MoveL 10412 to (233.6, 37.71, 144.49) mm, rotated rx 180 ry 0 rz 180 deg; joints [-18.033, 5.361, 78.709, 72.392, 18.952, -71.45]
  MoveL 10413 to (233.6, 37.71, 144.49) mm, rotated rx 180 ry 0 rz 180 deg; joints [-18.033, 5.361, 78.709, 72.392, 18.952, -71.45]
  Call Extruder(591.82547)
  MoveL 10414 to (233.9, 37.89, 144.49) mm, rotated rx 180 ry 0 rz 180 deg; joints [-18.041, 5.417, 78.648, 72.387, 18.961, -71.444]
  MoveL 10415 to (233.9, 37.89, 144.49) mm, rotated rx 180 ry 0 rz 180 deg; joints [-18.041, 5.417, 78.648, 72.387, 18.961, -71.444]
  Call Extruder(592.03398)
  MoveL 10416 to (234.21, 38.07, 144.49) mm, rotated rx -180 ry 0 rz 180 deg; joints [-18.049, 5.473, 78.587, 72.381, 18.971, -71.437]
  MoveL 10417 to (234.21, 38.07, 144.49) mm, rotated rx -180 ry 0 rz 180 deg; joints [-18.049, 5.473, 78.587, 72.381, 18.971, -71.437]
  Call Extruder(592.21352)
  MoveL 10418 to (234.45, 38.24, 144.49) mm, rotated rx 180 ry 0 rz 180 deg; joints [-18.06, 5.519, 78.536, 72.38, 18.982, -71.434]
  MoveL 10419 to (234.45, 38.24, 144.49) mm, rotated rx 180 ry 0 rz 180 deg; joints [-18.06, 5.519, 78.536, 72.38, 18.982, -71.434]
  Call Extruder(592.54693)
  MoveL 10420 to (234.9, 38.57, 144.49) mm, rotated rx -180 ry 0 rz -180 deg; joints [-18.079, 5.606, 78.442, 72.377, 19.003, -71.43]
  MoveL 10421 to (234.9, 38.57, 144.49) mm, rotated rx -180 ry 0 rz -180 deg; joints [-18.079, 5.606, 78.442, 72.377, 19.003, -71.43]
  Call Extruder(592.88153)
  MoveL 10422 to (235.35, 38.9, 144.49) mm, rotated rx 180 ry 0 rz 180 deg; joints [-18.099, 5.693, 78.347, 72.375, 19.024, -71.424]
  Call Extruder(593.70948)
  MoveL 10423 to (236.39, 39.81, 144.49) mm, rotated rx 180 ry 0 rz 180 deg; joints [-18.16, 5.9, 78.121, 72.381, 19.088, -71.425]
  Call Extruder(594.53743)
  MoveL 10424 to (237.3, 40.85, 144.49) mm, rotated rx 180 ry 0 rz 180 deg; joints [-18.24, 6.095, 77.907, 72.406, 19.169, -71.442]
  Call Extruder(594.70473)
  MoveL 10425 to (237.47, 41.07, 144.49) mm, rotated rx -180 ry 0 rz 180 deg; joints [-18.258, 6.132, 77.866, 72.414, 19.187, -71.449]
  MoveL 10426 to (237.47, 41.07, 144.49) mm, rotated rx -180 ry 0 rz 180 deg; joints [-18.258, 6.132, 77.866, 72.414, 19.187, -71.449]
  Call Extruder(595.03814)
  MoveL 10427 to (237.79, 41.52, 144.49) mm, rotated rx 180 ry 0 rz 180 deg; joints [-18.295, 6.206, 77.785, 72.429, 19.224, -71.461]
  MoveL 10428 to (237.79, 41.52, 144.49) mm, rotated rx 180 ry 0 rz 180 deg; joints [-18.295, 6.206, 77.785, 72.429, 19.224, -71.461]
  Call Extruder(595.37037)
  MoveL 10429 to (238.12, 41.98, 144.49) mm, rotated rx 180 ry 0 rz 180 deg; joints [-18.332, 6.28, 77.703, 72.444, 19.262, -71.472]
  MoveL 10430 to (238.12, 41.98, 144.49) mm, rotated rx 180 ry 0 rz 180 deg; joints [-18.332, 6.28, 77.703, 72.444, 19.262, -71.472]
  Call Extruder(595.48807)
  MoveL 10431 to (238.22, 42.15, 144.49) mm, rotated rx -180 ry 0 rz 180 deg; joints [-18.346, 6.305, 77.676, 72.452, 19.276, -71.479]
  MoveL 10432 to (238.22, 42.15, 144.49) mm, rotated rx -180 ry 0 rz 180 deg; joints [-18.346, 6.305, 77.676, 72.452, 19.276, -71.479]
  Call Extruder(595.69580)
  MoveL 10433 to (238.4, 42.45, 144.49) mm, rotated rx 180 ry 0 rz 180 deg; joints [-18.373, 6.348, 77.628, 72.465, 19.303, -71.49]
  MoveL 10434 to (238.4, 42.45, 144.49) mm, rotated rx 180 ry 0 rz 180 deg; joints [-18.373, 6.348, 77.628, 72.465, 19.303, -71.49]
  Call Extruder(595.90274)
  MoveL 10435 to (238.57, 42.75, 144.49) mm, rotated rx 180 ry 0 rz 180 deg; joints [-18.399, 6.391, 77.581, 72.478, 19.329, -71.501]
  MoveL 10436 to (238.57, 42.75, 144.49) mm, rotated rx 180 ry 0 rz 180 deg; joints [-18.399, 6.391, 77.581, 72.478, 19.329, -71.501]
  Call Extruder(596.10891)
  MoveL 10437 to (238.75, 43.06, 144.49) mm, rotated rx 180 ry 0 rz 180 deg; joints [-18.425, 6.434, 77.534, 72.491, 19.355, -71.512]
  MoveL 10438 to (238.75, 43.06, 144.49) mm, rotated rx 180 ry 0 rz 180 deg; joints [-18.425, 6.434, 77.534, 72.491, 19.355, -71.512]
  Call Extruder(596.29060)
  MoveL 10439 to (238.89, 43.34, 144.49) mm, rotated rx 180 ry 0 rz 180 deg; joints [-18.45, 6.47, 77.493, 72.504, 19.379, -71.523]
  MoveL 10440 to (238.89, 43.34, 144.49) mm, rotated rx 180 ry 0 rz 180 deg; joints [-18.45, 6.47, 77.493, 72.504, 19.379, -71.523]
  Call Extruder(596.44861)
  MoveL 10441 to (239, 43.58, 144.49) mm, rotated rx 180 ry 0 rz 180 deg; joints [-18.472, 6.5, 77.461, 72.518, 19.402, -71.534]
  MoveL 10442 to (239, 43.58, 144.49) mm, rotated rx 180 ry 0 rz 180 deg; joints [-18.472, 6.5, 77.461, 72.518, 19.402, -71.534]
  Call Extruder(596.60601)
  MoveL 10443 to (239.11, 43.83, 144.49) mm, rotated rx -180 ry 0 rz -180 deg; joints [-18.495, 6.529, 77.428, 72.531, 19.424, -71.546]
  MoveL 10444 to (239.11, 43.83, 144.49) mm, rotated rx -180 ry 0 rz -180 deg; joints [-18.495, 6.529, 77.428, 72.531, 19.424, -71.546]
  Call Extruder(596.78872)
  MoveL 10445 to (239.23, 44.12, 144.49) mm, rotated rx -180 ry 0 rz 180 deg; joints [-18.522, 6.563, 77.39, 72.547, 19.451, -71.56]
  MoveL 10446 to (239.23, 44.12, 144.49) mm, rotated rx -180 ry 0 rz 180 deg; joints [-18.522, 6.563, 77.39, 72.547, 19.451, -71.56]
  Call Extruder(596.97068)
  MoveL 10447 to (239.35, 44.42, 144.49) mm, rotated rx -180 ry 0 rz 180 deg; joints [-18.549, 6.598, 77.353, 72.562, 19.477, -71.573]
  MoveL 10448 to (239.35, 44.42, 144.49) mm, rotated rx -180 ry 0 rz 180 deg; joints [-18.549, 6.598, 77.353, 72.562, 19.477, -71.573]
  Call Extruder(597.11801)
  MoveL 10449 to (239.44, 44.66, 144.49) mm, rotated rx 180 ry 0 rz -180 deg; joints [-18.571, 6.624, 77.323, 72.576, 19.499, -71.585]
  MoveL 10450 to (239.44, 44.66, 144.49) mm, rotated rx 180 ry 0 rz -180 deg; joints [-18.571, 6.624, 77.323, 72.576, 19.499, -71.585]
  Call Extruder(597.23124)
  MoveL 10451 to (239.5, 44.85, 144.49) mm, rotated rx 180 ry 0 rz 180 deg; joints [-18.589, 6.644, 77.301, 72.587, 19.517, -71.595]
  MoveL 10452 to (239.5, 44.85, 144.49) mm, rotated rx 180 ry 0 rz 180 deg; joints [-18.589, 6.644, 77.301, 72.587, 19.517, -71.595]
  Call Extruder(597.34404)
  MoveL 10453 to (239.56, 45.03, 144.49) mm, rotated rx 180 ry 0 rz 180 deg; joints [-18.607, 6.663, 77.28, 72.598, 19.535, -71.605]
  MoveL 10454 to (239.56, 45.03, 144.49) mm, rotated rx 180 ry 0 rz 180 deg; joints [-18.607, 6.663, 77.28, 72.598, 19.535, -71.605]
  Call Extruder(597.45638)
  MoveL 10455 to (239.62, 45.22, 144.49) mm, rotated rx -180 ry 0 rz 180 deg; joints [-18.625, 6.683, 77.258, 72.609, 19.552, -71.615]
  MoveL 10456 to (239.62, 45.22, 144.49) mm, rotated rx -180 ry 0 rz 180 deg; joints [-18.625, 6.683, 77.258, 72.609, 19.552, -71.615]
  Call Extruder(597.56829)
  MoveL 10457 to (239.68, 45.41, 144.49) mm, rotated rx 180 ry 0 rz -180 deg; joints [-18.642, 6.702, 77.237, 72.62, 19.57, -71.625]
  MoveL 10458 to (239.68, 45.41, 144.49) mm, rotated rx 180 ry 0 rz -180 deg; joints [-18.642, 6.702, 77.237, 72.62, 19.57, -71.625]
  Call Extruder(597.68969)
  MoveL 10459 to (239.75, 45.62, 144.49) mm, rotated rx 180 ry 0 rz 180 deg; joints [-18.662, 6.723, 77.213, 72.633, 19.589, -71.635]
  MoveL 10460 to (239.75, 45.62, 144.49) mm, rotated rx 180 ry 0 rz 180 deg; joints [-18.662, 6.723, 77.213, 72.633, 19.589, -71.635]
  Call Extruder(597.82048)
  MoveL 10461 to (239.81, 45.84, 144.49) mm, rotated rx 180 ry 0 rz 180 deg; joints [-18.683, 6.745, 77.189, 72.646, 19.61, -71.647]
  MoveL 10462 to (239.81, 45.84, 144.49) mm, rotated rx 180 ry 0 rz 180 deg; joints [-18.683, 6.745, 77.189, 72.646, 19.61, -71.647]
  Call Extruder(597.95070)
  MoveL 10463 to (239.88, 46.06, 144.49) mm, rotated rx -180 ry 0 rz 180 deg; joints [-18.705, 6.768, 77.164, 72.66, 19.631, -71.659]
  MoveL 10464 to (239.88, 46.06, 144.49) mm, rotated rx -180 ry 0 rz 180 deg; joints [-18.705, 6.768, 77.164, 72.66, 19.631, -71.659]
  Call Extruder(598.08036)
  MoveL 10465 to (239.95, 46.29, 144.49) mm, rotated rx 180 ry 0 rz 180 deg; joints [-18.726, 6.79, 77.139, 72.673, 19.652, -71.671]
  MoveL 10466 to (239.95, 46.29, 144.49) mm, rotated rx 180 ry 0 rz 180 deg; joints [-18.726, 6.79, 77.139, 72.673, 19.652, -71.671]
  Call Extruder(598.20946)
  MoveL 10467 to (240.02, 46.51, 144.49) mm, rotated rx 180 ry 0 rz 180 deg; joints [-18.747, 6.812, 77.114, 72.686, 19.673, -71.683]
  MoveL 10468 to (240.02, 46.51, 144.49) mm, rotated rx 180 ry 0 rz 180 deg; joints [-18.747, 6.812, 77.114, 72.686, 19.673, -71.683]
  Call Extruder(598.32451)
  MoveL 10469 to (240.06, 46.72, 144.49) mm, rotated rx 180 ry 0 rz 180 deg; joints [-18.767, 6.83, 77.095, 72.7, 19.692, -71.695]
  MoveL 10470 to (240.06, 46.72, 144.49) mm, rotated rx 180 ry 0 rz 180 deg; joints [-18.767, 6.83, 77.095, 72.7, 19.692, -71.695]
  Call Extruder(598.43912)
  MoveL 10471 to (240.11, 46.92, 144.49) mm, rotated rx 180 ry 0 rz 180 deg; joints [-18.787, 6.848, 77.075, 72.713, 19.712, -71.707]
  MoveL 10472 to (240.11, 46.92, 144.49) mm, rotated rx 180 ry 0 rz 180 deg; joints [-18.787, 6.848, 77.075, 72.713, 19.712, -71.707]
  Call Extruder(598.55327)
  MoveL 10473 to (240.15, 47.12, 144.49) mm, rotated rx 180 ry 0 rz 180 deg; joints [-18.807, 6.866, 77.055, 72.727, 19.732, -71.719]
  MoveL 10474 to (240.15, 47.12, 144.49) mm, rotated rx 180 ry 0 rz 180 deg; joints [-18.807, 6.866, 77.055, 72.727, 19.732, -71.719]
  Call Extruder(598.66696)
  MoveL 10475 to (240.2, 47.33, 144.49) mm, rotated rx 180 ry 0 rz 180 deg; joints [-18.827, 6.884, 77.035, 72.74, 19.751, -71.731]
  MoveL 10476 to (240.2, 47.33, 144.49) mm, rotated rx 180 ry 0 rz 180 deg; joints [-18.827, 6.884, 77.035, 72.74, 19.751, -71.731]
  Call Extruder(598.79237)
  MoveL 10477 to (240.24, 47.55, 144.49) mm, rotated rx 180 ry 0 rz 180 deg; joints [-18.85, 6.903, 77.014, 72.755, 19.773, -71.744]
  MoveL 10478 to (240.24, 47.55, 144.49) mm, rotated rx 180 ry 0 rz 180 deg; joints [-18.85, 6.903, 77.014, 72.755, 19.773, -71.744]
  Call Extruder(598.92935)
  MoveL 10479 to (240.29, 47.8, 144.49) mm, rotated rx 180 ry 0 rz -180 deg; joints [-18.874, 6.924, 76.99, 72.771, 19.797, -71.759]
  MoveL 10480 to (240.29, 47.8, 144.49) mm, rotated rx 180 ry 0 rz -180 deg; joints [-18.874, 6.924, 76.99, 72.771, 19.797, -71.759]
  Call Extruder(599.06572)
  MoveL 10481 to (240.34, 48.05, 144.49) mm, rotated rx 180 ry 0 rz 180 deg; joints [-18.899, 6.945, 76.967, 72.788, 19.821, -71.774]
  MoveL 10482 to (240.34, 48.05, 144.49) mm, rotated rx 180 ry 0 rz 180 deg; joints [-18.899, 6.945, 76.967, 72.788, 19.821, -71.774]
  Call Extruder(599.20147)
  MoveL 10483 to (240.39, 48.3, 144.49) mm, rotated rx 180 ry 0 rz 180 deg; joints [-18.923, 6.966, 76.943, 72.804, 19.845, -71.788]
  MoveL 10484 to (240.39, 48.3, 144.49) mm, rotated rx 180 ry 0 rz 180 deg; joints [-18.923, 6.966, 76.943, 72.804, 19.845, -71.788]
  Call Extruder(599.33662)
  MoveL 10485 to (240.44, 48.55, 144.49) mm, rotated rx 180 ry 0 rz 180 deg; joints [-18.948, 6.987, 76.92, 72.821, 19.869, -71.803]
  MoveL 10486 to (240.44, 48.55, 144.49) mm, rotated rx 180 ry 0 rz 180 deg; joints [-18.948, 6.987, 76.92, 72.821, 19.869, -71.803]
  Call Extruder(599.47116)
  MoveL 10487 to (240.49, 48.8, 144.49) mm, rotated rx 180 ry 0 rz 180 deg; joints [-18.973, 7.008, 76.897, 72.837, 19.893, -71.817]
  MoveL 10488 to (240.49, 48.8, 144.49) mm, rotated rx 180 ry 0 rz 180 deg; joints [-18.973, 7.008, 76.897, 72.837, 19.893, -71.817]
  Call Extruder(599.60508)
  MoveL 10489 to (240.54, 49.05, 144.49) mm, rotated rx 180 ry 0 rz 180 deg; joints [-18.997, 7.029, 76.873, 72.853, 19.917, -71.832]
  MoveL 10490 to (240.54, 49.05, 144.49) mm, rotated rx 180 ry 0 rz 180 deg; joints [-18.997, 7.029, 76.873, 72.853, 19.917, -71.832]
  Call Extruder(599.75295)
  MoveL 10491 to (240.59, 49.33, 144.49) mm, rotated rx 180 ry 0 rz 180 deg; joints [-19.025, 7.052, 76.848, 72.871, 19.944, -71.848]
  MoveL 10492 to (240.59, 49.33, 144.49) mm, rotated rx 180 ry 0 rz 180 deg; joints [-19.025, 7.052, 76.848, 72.871, 19.944, -71.848]
  Call Extruder(599.91470)
  MoveL 10493 to (240.64, 49.63, 144.49) mm, rotated rx 180 ry 0 rz 180 deg; joints [-19.055, 7.076, 76.821, 72.892, 19.974, -71.867]
  MoveL 10494 to (240.64, 49.63, 144.49) mm, rotated rx 180 ry 0 rz 180 deg; joints [-19.055, 7.076, 76.821, 72.892, 19.974, -71.867]
  Call Extruder(600.07571)
  MoveL 10495 to (240.69, 49.94, 144.49) mm, rotated rx 180 ry 0 rz 180 deg; joints [-19.086, 7.1, 76.794, 72.912, 20.004, -71.885]
  MoveL 10496 to (240.69, 49.94, 144.49) mm, rotated rx 180 ry 0 rz 180 deg; joints [-19.086, 7.1, 76.794, 72.912, 20.004, -71.885]
  Call Extruder(600.23600)
  MoveL 10497 to (240.74, 50.24, 144.49) mm, rotated rx 180 ry 0 rz 180 deg; joints [-19.116, 7.124, 76.768, 72.933, 20.033, -71.903]
  MoveL 10498 to (240.74, 50.24, 144.49) mm, rotated rx 180 ry 0 rz 180 deg; joints [-19.116, 7.124, 76.768, 72.933, 20.033, -71.903]
  Call Extruder(600.39556)
  MoveL 10499 to (240.78, 50.55, 144.49) mm, rotated rx 180 ry 0 rz 180 deg; joints [-19.146, 7.148, 76.741, 72.953, 20.063, -71.921]
  MoveL 10500 to (240.78, 50.55, 144.49) mm, rotated rx 180 ry 0 rz 180 deg; joints [-19.146, 7.148, 76.741, 72.953, 20.063, -71.921]
  Call Extruder(600.55440)
  MoveL 10501 to (240.83, 50.86, 144.49) mm, rotated rx 180 ry 0 rz 180 deg; joints [-19.177, 7.172, 76.714, 72.973, 20.093, -71.939]
  MoveL 10502 to (240.83, 50.86, 144.49) mm, rotated rx 180 ry 0 rz 180 deg; joints [-19.177, 7.172, 76.714, 72.973, 20.093, -71.939]
  Call Extruder(600.73307)
  MoveL 10503 to (240.88, 51.2, 144.49) mm, rotated rx 180 ry 0 rz 180 deg; joints [-19.212, 7.199, 76.684, 72.997, 20.127, -71.96]
  MoveL 10504 to (240.88, 51.2, 144.49) mm, rotated rx 180 ry 0 rz 180 deg; joints [-19.212, 7.199, 76.684, 72.997, 20.127, -71.96]
  Call Extruder(600.93151)
  MoveL 10505 to (240.92, 51.59, 144.49) mm, rotated rx 180 ry 0 rz 180 deg; joints [-19.251, 7.227, 76.653, 73.023, 20.165, -71.984]
  MoveL 10506 to (240.92, 51.59, 144.49) mm, rotated rx 180 ry 0 rz 180 deg; joints [-19.251, 7.227, 76.653, 73.023, 20.165, -71.984]
  Call Extruder(601.12909)
  MoveL 10507 to (240.97, 51.98, 144.49) mm, rotated rx 180 ry 0 rz 180 deg; joints [-19.29, 7.255, 76.621, 73.05, 20.203, -72.008]
  MoveL 10508 to (240.97, 51.98, 144.49) mm, rotated rx 180 ry 0 rz 180 deg; joints [-19.29, 7.255, 76.621, 73.05, 20.203, -72.008]
  Call Extruder(601.32579)
  MoveL 10509 to (241.02, 52.36, 144.49) mm, rotated rx 180 ry 0 rz 180 deg; joints [-19.329, 7.284, 76.59, 73.076, 20.241, -72.031]
  MoveL 10510 to (241.02, 52.36, 144.49) mm, rotated rx 180 ry 0 rz 180 deg; joints [-19.329, 7.284, 76.59, 73.076, 20.241, -72.031]
  Call Extruder(601.52163)
  MoveL 10511 to (241.06, 52.75, 144.49) mm, rotated rx -180 ry 0 rz 180 deg; joints [-19.368, 7.312, 76.558, 73.102, 20.279, -72.055]
  MoveL 10512 to (241.06, 52.75, 144.49) mm, rotated rx -180 ry 0 rz 180 deg; joints [-19.368, 7.312, 76.558, 73.102, 20.279, -72.055]
  Call Extruder(601.81707)
  MoveL 10513 to (241.11, 53.34, 144.49) mm, rotated rx 180 ry 0 rz -180 deg; joints [-19.428, 7.352, 76.514, 73.143, 20.338, -72.092]
  MoveL 10514 to (241.11, 53.34, 144.49) mm, rotated rx 180 ry 0 rz -180 deg; joints [-19.428, 7.352, 76.514, 73.143, 20.338, -72.092]
  Call Extruder(602.11118)
  MoveL 10515 to (241.15, 53.93, 144.49) mm, rotated rx 180 ry 0 rz 180 deg; joints [-19.488, 7.391, 76.469, 73.184, 20.397, -72.129]
  MoveL 10516 to (241.15, 53.93, 144.49) mm, rotated rx 180 ry 0 rz 180 deg; joints [-19.488, 7.391, 76.469, 73.184, 20.397, -72.129]
  Call Extruder(602.40395)
  MoveL 10517 to (241.2, 54.52, 144.49) mm, rotated rx 180 ry 0 rz 180 deg; joints [-19.548, 7.431, 76.424, 73.224, 20.455, -72.165]
  MoveL 10518 to (241.2, 54.52, 144.49) mm, rotated rx 180 ry 0 rz 180 deg; joints [-19.548, 7.431, 76.424, 73.224, 20.455, -72.165]
  Call Extruder(602.97740)
  MoveL 10519 to (241.25, 55.68, 144.49) mm, rotated rx -180 ry 0 rz 180 deg; joints [-19.668, 7.503, 76.344, 73.307, 20.572, -72.239]
  MoveL 10520 to (241.25, 55.68, 144.49) mm, rotated rx -180 ry 0 rz 180 deg; joints [-19.668, 7.503, 76.344, 73.307, 20.572, -72.239]
  Call Extruder(603.69124)
  MoveL 10521 to (241.29, 57.14, 144.49) mm, rotated rx -180 ry 0 rz 180 deg; joints [-19.819, 7.59, 76.246, 73.41, 20.718, -72.332]
  Call Extruder(645.75613)
  MoveL 10522 to (241.29, 142.86, 144.49) mm, rotated rx -180 ry 0 rz 180 deg; joints [-28.232, 13.571, 69.243, 76.885, 29.059, -75.075]
  Call Extruder(646.18456)
  MoveL 10523 to (241.27, 143.74, 144.49) mm, rotated rx -180 ry 0 rz 180 deg; joints [-28.313, 13.641, 69.157, 76.9, 29.141, -75.081]
  MoveL 10524 to (241.27, 143.74, 144.49) mm, rotated rx -180 ry 0 rz 180 deg; joints [-28.313, 13.641, 69.157, 76.9, 29.141, -75.081]
  Call Extruder(646.75801)
  MoveL 10525 to (241.22, 144.9, 144.49) mm, rotated rx 180 ry 0 rz 180 deg; joints [-28.421, 13.732, 69.046, 76.922, 29.25, -75.091]
  MoveL 10526 to (241.22, 144.9, 144.49) mm, rotated rx 180 ry 0 rz 180 deg; joints [-28.421, 13.732, 69.046, 76.922, 29.25, -75.091]
  Call Extruder(647.19234)
  MoveL 10527 to (241.18, 145.77, 144.49) mm, rotated rx -180 ry 0 rz -180 deg; joints [-28.503, 13.799, 68.964, 76.94, 29.333, -75.099]
  MoveL 10528 to (241.18, 145.77, 144.49) mm, rotated rx -180 ry 0 rz -180 deg; joints [-28.503, 13.799, 68.964, 76.94, 29.333, -75.099]
  Call Extruder(647.48645)
  MoveL 10529 to (241.13, 146.36, 144.49) mm, rotated rx -180 ry 0 rz -180 deg; joints [-28.559, 13.841, 68.912, 76.953, 29.389, -75.106]
  MoveL 10530 to (241.13, 146.36, 144.49) mm, rotated rx -180 ry 0 rz -180 deg; joints [-28.559, 13.841, 68.912, 76.953, 29.389, -75.106]
  Call Extruder(647.78189)
  MoveL 10531 to (241.09, 146.95, 144.49) mm, rotated rx -180 ry 0 rz -180 deg; joints [-28.615, 13.884, 68.86, 76.965, 29.445, -75.112]
  MoveL 10532 to (241.09, 146.95, 144.49) mm, rotated rx -180 ry 0 rz -180 deg; joints [-28.615, 13.884, 68.86, 76.965, 29.445, -75.112]
  Call Extruder(648.02815)
  MoveL 10533 to (241.04, 147.44, 144.49) mm, rotated rx 180 ry 0 rz 180 deg; joints [-28.662, 13.919, 68.818, 76.976, 29.492, -75.118]
  MoveL 10534 to (241.04, 147.44, 144.49) mm, rotated rx 180 ry 0 rz 180 deg; joints [-28.662, 13.919, 68.818, 76.976, 29.492, -75.118]
  Call Extruder(648.22485)
  MoveL 10535 to (240.99, 147.83, 144.49) mm, rotated rx -180 ry 0 rz 180 deg; joints [-28.7, 13.945, 68.786, 76.986, 29.53, -75.124]
  MoveL 10536 to (240.99, 147.83, 144.49) mm, rotated rx -180 ry 0 rz 180 deg; joints [-28.7, 13.945, 68.786, 76.986, 29.53, -75.124]
  Call Extruder(648.42243)
  MoveL 10537 to (240.95, 148.22, 144.49) mm, rotated rx 180 ry 0 rz 180 deg; joints [-28.737, 13.97, 68.754, 76.995, 29.567, -75.129]
  MoveL 10538 to (240.95, 148.22, 144.49) mm, rotated rx 180 ry 0 rz 180 deg; joints [-28.737, 13.97, 68.754, 76.995, 29.567, -75.129]
  Call Extruder(648.62087)
  MoveL 10539 to (240.9, 148.6, 144.49) mm, rotated rx 180 ry 0 rz 180 deg; joints [-28.774, 13.996, 68.722, 77.005, 29.605, -75.135]
  MoveL 10540 to (240.9, 148.6, 144.49) mm, rotated rx 180 ry 0 rz 180 deg; joints [-28.774, 13.996, 68.722, 77.005, 29.605, -75.135]
  Call Extruder(648.82018)
  MoveL 10541 to (240.86, 148.99, 144.49) mm, rotated rx 180 ry 0 rz 180 deg; joints [-28.812, 14.022, 68.691, 77.014, 29.642, -75.14]
  MoveL 10542 to (240.86, 148.99, 144.49) mm, rotated rx 180 ry 0 rz 180 deg; joints [-28.812, 14.022, 68.691, 77.014, 29.642, -75.14]
  Call Extruder(648.97901)
  MoveL 10543 to (240.81, 149.3, 144.49) mm, rotated rx 180 ry 0 rz 180 deg; joints [-28.842, 14.041, 68.668, 77.022, 29.672, -75.145]
  MoveL 10544 to (240.81, 149.3, 144.49) mm, rotated rx 180 ry 0 rz 180 deg; joints [-28.842, 14.041, 68.668, 77.022, 29.672, -75.145]
  Call Extruder(649.13857)
  MoveL 10545 to (240.76, 149.6, 144.49) mm, rotated rx 180 ry 0 rz 180 deg; joints [-28.872, 14.06, 68.645, 77.031, 29.703, -75.15]
  MoveL 10546 to (240.76, 149.6, 144.49) mm, rotated rx 180 ry 0 rz 180 deg; joints [-28.872, 14.06, 68.645, 77.031, 29.703, -75.15]
  Call Extruder(649.29886)
  MoveL 10547 to (240.71, 149.91, 144.49) mm, rotated rx 180 ry 0 rz 180 deg; joints [-28.902, 14.078, 68.622, 77.039, 29.732, -75.155]
  MoveL 10548 to (240.71, 149.91, 144.49) mm, rotated rx 180 ry 0 rz 180 deg; joints [-28.902, 14.078, 68.622, 77.039, 29.732, -75.155]
  Call Extruder(649.45987)
  MoveL 10549 to (240.66, 150.21, 144.49) mm, rotated rx 180 ry 0 rz -180 deg; joints [-28.932, 14.097, 68.599, 77.047, 29.763, -75.161]
  MoveL 10550 to (240.66, 150.21, 144.49) mm, rotated rx 180 ry 0 rz -180 deg; joints [-28.932, 14.097, 68.599, 77.047, 29.763, -75.161]
  Call Extruder(649.62162)
  MoveL 10551 to (240.61, 150.52, 144.49) mm, rotated rx 180 ry 0 rz 180 deg; joints [-28.962, 14.116, 68.576, 77.056, 29.793, -75.166]
  MoveL 10552 to (240.61, 150.52, 144.49) mm, rotated rx 180 ry 0 rz 180 deg; joints [-28.962, 14.116, 68.576, 77.056, 29.793, -75.166]
  Call Extruder(649.78409)
  MoveL 10553 to (240.57, 150.83, 144.49) mm, rotated rx -180 ry 0 rz 180 deg; joints [-28.993, 14.135, 68.553, 77.064, 29.823, -75.171]
  MoveL 10554 to (240.57, 150.83, 144.49) mm, rotated rx -180 ry 0 rz 180 deg; joints [-28.993, 14.135, 68.553, 77.064, 29.823, -75.171]
  Call Extruder(649.91802)
  MoveL 10555 to (240.52, 151.08, 144.49) mm, rotated rx 180 ry 0 rz 180 deg; joints [-29.017, 14.149, 68.535, 77.071, 29.848, -75.176]
  MoveL 10556 to (240.52, 151.08, 144.49) mm, rotated rx 180 ry 0 rz 180 deg; joints [-29.017, 14.149, 68.535, 77.071, 29.848, -75.176]
  Call Extruder(650.05255)
  MoveL 10557 to (240.47, 151.32, 144.49) mm, rotated rx 180 ry 0 rz 180 deg; joints [-29.043, 14.162, 68.519, 77.079, 29.872, -75.181]
  MoveL 10558 to (240.47, 151.32, 144.49) mm, rotated rx 180 ry 0 rz 180 deg; joints [-29.043, 14.162, 68.519, 77.079, 29.872, -75.181]
  Call Extruder(650.18770)
  MoveL 10559 to (240.42, 151.57, 144.49) mm, rotated rx -180 ry 0 rz 180 deg; joints [-29.067, 14.176, 68.502, 77.086, 29.897, -75.186]
  MoveL 10560 to (240.42, 151.57, 144.49) mm, rotated rx -180 ry 0 rz 180 deg; joints [-29.067, 14.176, 68.502, 77.086, 29.897, -75.186]
  Call Extruder(650.32346)
  MoveL 10561 to (240.37, 151.82, 144.49) mm, rotated rx 180 ry 0 rz 180 deg; joints [-29.092, 14.19, 68.485, 77.094, 29.922, -75.19]
  MoveL 10562 to (240.37, 151.82, 144.49) mm, rotated rx 180 ry 0 rz 180 deg; joints [-29.092, 14.19, 68.485, 77.094, 29.922, -75.19]
  Call Extruder(650.45983)
  MoveL 10563 to (240.32, 152.07, 144.49) mm, rotated rx 180 ry 0 rz 180 deg; joints [-29.117, 14.204, 68.468, 77.101, 29.947, -75.195]
  MoveL 10564 to (240.32, 152.07, 144.49) mm, rotated rx 180 ry 0 rz 180 deg; joints [-29.117, 14.204, 68.468, 77.101, 29.947, -75.195]
  Call Extruder(650.59680)
  MoveL 10565 to (240.27, 152.32, 144.49) mm, rotated rx 180 ry 0 rz 180 deg; joints [-29.142, 14.218, 68.45, 77.108, 29.972, -75.2]
  MoveL 10566 to (240.27, 152.32, 144.49) mm, rotated rx 180 ry 0 rz 180 deg; joints [-29.142, 14.218, 68.45, 77.108, 29.972, -75.2]
  Call Extruder(650.73439)
  MoveL 10567 to (240.22, 152.57, 144.49) mm, rotated rx 180 ry 0 rz 180 deg; joints [-29.167, 14.232, 68.433, 77.116, 29.997, -75.205]
  MoveL 10568 to (240.22, 152.57, 144.49) mm, rotated rx 180 ry 0 rz 180 deg; joints [-29.167, 14.232, 68.433, 77.116, 29.997, -75.205]
  Call Extruder(650.84809)
  MoveL 10569 to (240.17, 152.77, 144.49) mm, rotated rx 180 ry 0 rz -180 deg; joints [-29.188, 14.243, 68.42, 77.122, 30.017, -75.209]
  MoveL 10570 to (240.17, 152.77, 144.49) mm, rotated rx 180 ry 0 rz -180 deg; joints [-29.188, 14.243, 68.42, 77.122, 30.017, -75.209]
  Call Extruder(650.96224)
  MoveL 10571 to (240.13, 152.98, 144.49) mm, rotated rx 180 ry 0 rz 180 deg; joints [-29.209, 14.253, 68.407, 77.128, 30.038, -75.213]
  MoveL 10572 to (240.13, 152.98, 144.49) mm, rotated rx 180 ry 0 rz 180 deg; joints [-29.209, 14.253, 68.407, 77.128, 30.038, -75.213]
  Call Extruder(651.07684)
  MoveL 10573 to (240.08, 153.18, 144.49) mm, rotated rx 180 ry 0 rz 180 deg; joints [-29.229, 14.264, 68.393, 77.135, 30.058, -75.218]
  MoveL 10574 to (240.08, 153.18, 144.49) mm, rotated rx 180 ry 0 rz 180 deg; joints [-29.229, 14.264, 68.393, 77.135, 30.058, -75.218]
  Call Extruder(651.19190)
  MoveL 10575 to (240.04, 153.39, 144.49) mm, rotated rx -180 ry 0 rz 180 deg; joints [-29.25, 14.275, 68.38, 77.141, 30.079, -75.222]
  MoveL 10576 to (240.04, 153.39, 144.49) mm, rotated rx -180 ry 0 rz 180 deg; joints [-29.25, 14.275, 68.38, 77.141, 30.079, -75.222]
  Call Extruder(651.31412)
  MoveL 10577 to (239.98, 153.6, 144.49) mm, rotated rx 180 ry 0 rz 180 deg; joints [-29.272, 14.285, 68.368, 77.148, 30.101, -75.227]
  MoveL 10578 to (239.98, 153.6, 144.49) mm, rotated rx 180 ry 0 rz 180 deg; joints [-29.272, 14.285, 68.368, 77.148, 30.101, -75.227]
  Call Extruder(651.44378)
  MoveL 10579 to (239.92, 153.82, 144.49) mm, rotated rx 180 ry 0 rz 180 deg; joints [-29.296, 14.294, 68.357, 77.157, 30.124, -75.234]
  MoveL 10580 to (239.92, 153.82, 144.49) mm, rotated rx 180 ry 0 rz 180 deg; joints [-29.296, 14.294, 68.357, 77.157, 30.124, -75.234]
  Call Extruder(651.57401)
  MoveL 10581 to (239.85, 154.05, 144.49) mm, rotated rx 180 ry 0 rz -180 deg; joints [-29.319, 14.303, 68.346, 77.165, 30.147, -75.24]
  MoveL 10582 to (239.85, 154.05, 144.49) mm, rotated rx 180 ry 0 rz -180 deg; joints [-29.319, 14.303, 68.346, 77.165, 30.147, -75.24]
  Call Extruder(651.70480)
  MoveL 10583 to (239.78, 154.27, 144.49) mm, rotated rx 180 ry 0 rz 180 deg; joints [-29.343, 14.312, 68.335, 77.174, 30.17, -75.246]
  MoveL 10584 to (239.78, 154.27, 144.49) mm, rotated rx 180 ry 0 rz 180 deg; joints [-29.343, 14.312, 68.335, 77.174, 30.17, -75.246]
  Call Extruder(651.83615)
  MoveL 10585 to (239.71, 154.5, 144.49) mm, rotated rx 180 ry 0 rz -180 deg; joints [-29.366, 14.321, 68.323, 77.182, 30.194, -75.252]
  MoveL 10586 to (239.71, 154.5, 144.49) mm, rotated rx 180 ry 0 rz -180 deg; joints [-29.366, 14.321, 68.323, 77.182, 30.194, -75.252]
  Call Extruder(651.94805)
  MoveL 10587 to (239.65, 154.68, 144.49) mm, rotated rx 180 ry 0 rz 180 deg; joints [-29.386, 14.328, 68.315, 77.19, 30.213, -75.258]
  MoveL 10588 to (239.65, 154.68, 144.49) mm, rotated rx 180 ry 0 rz 180 deg; joints [-29.386, 14.328, 68.315, 77.19, 30.213, -75.258]
  Call Extruder(652.06040)
  MoveL 10589 to (239.59, 154.87, 144.49) mm, rotated rx -180 ry 0 rz 180 deg; joints [-29.406, 14.335, 68.306, 77.197, 30.233, -75.264]
  MoveL 10590 to (239.59, 154.87, 144.49) mm, rotated rx -180 ry 0 rz 180 deg; joints [-29.406, 14.335, 68.306, 77.197, 30.233, -75.264]
  Call Extruder(652.17319)
  MoveL 10591 to (239.53, 155.06, 144.49) mm, rotated rx -180 ry 0 rz 180 deg; joints [-29.426, 14.342, 68.298, 77.204, 30.253, -75.269]
  MoveL 10592 to (239.53, 155.06, 144.49) mm, rotated rx -180 ry 0 rz 180 deg; joints [-29.426, 14.342, 68.298, 77.204, 30.253, -75.269]
  Call Extruder(652.28642)
  MoveL 10593 to (239.47, 155.25, 144.49) mm, rotated rx 180 ry 0 rz 180 deg; joints [-29.446, 14.349, 68.289, 77.212, 30.272, -75.275]
  MoveL 10594 to (239.47, 155.25, 144.49) mm, rotated rx 180 ry 0 rz 180 deg; joints [-29.446, 14.349, 68.289, 77.212, 30.272, -75.275]
  Call Extruder(652.40010)
  MoveL 10595 to (239.41, 155.44, 144.49) mm, rotated rx -180 ry 0 rz 180 deg; joints [-29.466, 14.356, 68.28, 77.219, 30.292, -75.28]
  MoveL 10596 to (239.41, 155.44, 144.49) mm, rotated rx -180 ry 0 rz 180 deg; joints [-29.466, 14.356, 68.28, 77.219, 30.292, -75.28]
  Call Extruder(652.58206)
  MoveL 10597 to (239.29, 155.73, 144.49) mm, rotated rx 180 ry 0 rz 180 deg; joints [-29.499, 14.363, 68.272, 77.233, 30.324, -75.291]
  MoveL 10598 to (239.29, 155.73, 144.49) mm, rotated rx 180 ry 0 rz 180 deg; joints [-29.499, 14.363, 68.272, 77.233, 30.324, -75.291]
  Call Extruder(652.76478)
  MoveL 10599 to (239.16, 156.02, 144.49) mm, rotated rx 180 ry 0 rz 180 deg; joints [-29.531, 14.37, 68.263, 77.246, 30.355, -75.302]
  MoveL 10600 to (239.16, 156.02, 144.49) mm, rotated rx 180 ry 0 rz 180 deg; joints [-29.531, 14.37, 68.263, 77.246, 30.355, -75.302]
  Call Extruder(652.93520)
  MoveL 10601 to (239.05, 156.29, 144.49) mm, rotated rx 180 ry 0 rz 180 deg; joints [-29.561, 14.376, 68.256, 77.259, 30.385, -75.313]
  MoveL 10602 to (239.05, 156.29, 144.49) mm, rotated rx 180 ry 0 rz 180 deg; joints [-29.561, 14.376, 68.256, 77.259, 30.385, -75.313]
  Call Extruder(653.09321)
  MoveL 10603 to (238.94, 156.54, 144.49) mm, rotated rx 180 ry 0 rz 180 deg; joints [-29.589, 14.381, 68.249, 77.271, 30.412, -75.322]
  MoveL 10604 to (238.94, 156.54, 144.49) mm, rotated rx 180 ry 0 rz 180 deg; joints [-29.589, 14.381, 68.249, 77.271, 30.412, -75.322]
  Call Extruder(653.25183)
  MoveL 10605 to (238.84, 156.79, 144.49) mm, rotated rx 180 ry 0 rz 180 deg; joints [-29.617, 14.387, 68.243, 77.283, 30.439, -75.332]
  MoveL 10606 to (238.84, 156.79, 144.49) mm, rotated rx 180 ry 0 rz 180 deg; joints [-29.617, 14.387, 68.243, 77.283, 30.439, -75.332]
  Call Extruder(653.45800)
  MoveL 10607 to (238.66, 157.09, 144.49) mm, rotated rx 180 ry 0 rz 180 deg; joints [-29.653, 14.386, 68.243, 77.301, 30.474, -75.347]
  MoveL 10608 to (238.66, 157.09, 144.49) mm, rotated rx 180 ry 0 rz 180 deg; joints [-29.653, 14.386, 68.243, 77.301, 30.474, -75.347]
  Call Extruder(653.66494)
  MoveL 10609 to (238.49, 157.4, 144.49) mm, rotated rx 180 ry 0 rz 180 deg; joints [-29.689, 14.386, 68.244, 77.319, 30.509, -75.363]
  MoveL 10610 to (238.49, 157.4, 144.49) mm, rotated rx 180 ry 0 rz 180 deg; joints [-29.689, 14.386, 68.244, 77.319, 30.509, -75.363]
  Call Extruder(653.87267)
  MoveL 10611 to (238.31, 157.7, 144.49) mm, rotated rx 180 ry 0 rz 180 deg; joints [-29.725, 14.386, 68.244, 77.337, 30.544, -75.379]
  MoveL 10612 to (238.31, 157.7, 144.49) mm, rotated rx 180 ry 0 rz 180 deg; joints [-29.725, 14.386, 68.244, 77.337, 30.544, -75.379]
  Call Extruder(654.08118)
  MoveL 10613 to (238.13, 158.01, 144.49) mm, rotated rx 180 ry 0 rz 180 deg; joints [-29.761, 14.385, 68.244, 77.355, 30.579, -75.394]
  MoveL 10614 to (238.13, 158.01, 144.49) mm, rotated rx 180 ry 0 rz 180 deg; joints [-29.761, 14.385, 68.244, 77.355, 30.579, -75.394]
  Call Extruder(654.26072)
  MoveL 10615 to (237.96, 158.25, 144.49) mm, rotated rx 180 ry 0 rz 180 deg; joints [-29.792, 14.38, 68.251, 77.373, 30.609, -75.41]
  MoveL 10616 to (237.96, 158.25, 144.49) mm, rotated rx 180 ry 0 rz 180 deg; joints [-29.792, 14.38, 68.251, 77.373, 30.609, -75.41]
  Call Extruder(654.59412)
  MoveL 10617 to (237.63, 158.7, 144.49) mm, rotated rx 180 ry 0 rz 180 deg; joints [-29.849, 14.369, 68.264, 77.405, 30.664, -75.439]
  MoveL 10618 to (237.63, 158.7, 144.49) mm, rotated rx 180 ry 0 rz 180 deg; joints [-29.849, 14.369, 68.264, 77.405, 30.664, -75.439]
  Call Extruder(654.92872)
  MoveL 10619 to (237.3, 159.15, 144.49) mm, rotated rx 180 ry 0 rz 180 deg; joints [-29.907, 14.358, 68.277, 77.437, 30.718, -75.468]
  Call Extruder(655.75669)
  MoveL 10620 to (236.39, 160.19, 144.49) mm, rotated rx 180 ry 0 rz -180 deg; joints [-30.046, 14.31, 68.337, 77.524, 30.851, -75.548]
  Call Extruder(656.58460)
  MoveL 10621 to (235.35, 161.1, 144.49) mm, rotated rx -180 ry 0 rz 180 deg; joints [-30.182, 14.232, 68.434, 77.619, 30.978, -75.639]
  Call Extruder(656.75191)
  MoveL 10622 to (235.13, 161.27, 144.49) mm, rotated rx 180 ry 0 rz -180 deg; joints [-30.208, 14.211, 68.458, 77.639, 31.003, -75.658]
  MoveL 10623 to (235.13, 161.27, 144.49) mm, rotated rx 180 ry 0 rz -180 deg; joints [-30.208, 14.211, 68.458, 77.639, 31.003, -75.658]
  Call Extruder(657.08534)
  MoveL 10624 to (234.68, 161.6, 144.49) mm, rotated rx 180 ry 0 rz 180 deg; joints [-30.261, 14.171, 68.508, 77.679, 31.052, -75.697]
  MoveL 10625 to (234.68, 161.6, 144.49) mm, rotated rx 180 ry 0 rz 180 deg; joints [-30.261, 14.171, 68.508, 77.679, 31.052, -75.697]
  Call Extruder(657.41758)
  MoveL 10626 to (234.23, 161.92, 144.49) mm, rotated rx 180 ry 0 rz 180 deg; joints [-30.314, 14.131, 68.557, 77.72, 31.101, -75.736]
  MoveL 10627 to (234.23, 161.92, 144.49) mm, rotated rx 180 ry 0 rz 180 deg; joints [-30.314, 14.131, 68.557, 77.72, 31.101, -75.736]
  Call Extruder(657.53524)
  MoveL 10628 to (234.05, 162.02, 144.49) mm, rotated rx 180 ry 0 rz 180 deg; joints [-30.331, 14.114, 68.578, 77.734, 31.118, -75.751]
  MoveL 10629 to (234.05, 162.02, 144.49) mm, rotated rx 180 ry 0 rz 180 deg; joints [-30.331, 14.114, 68.578, 77.734, 31.118, -75.751]
  Call Extruder(657.74297)
  MoveL 10630 to (233.75, 162.2, 144.49) mm, rotated rx 180 ry 0 rz 180 deg; joints [-30.363, 14.083, 68.616, 77.761, 31.147, -75.777]
  MoveL 10631 to (233.75, 162.2, 144.49) mm, rotated rx 180 ry 0 rz 180 deg; joints [-30.363, 14.083, 68.616, 77.761, 31.147, -75.777]
  Call Extruder(657.94993)
  MoveL 10632 to (233.45, 162.37, 144.49) mm, rotated rx 180 ry 0 rz 180 deg; joints [-30.394, 14.052, 68.654, 77.787, 31.176, -75.803]
  MoveL 10633 to (233.45, 162.37, 144.49) mm, rotated rx 180 ry 0 rz 180 deg; joints [-30.394, 14.052, 68.654, 77.787, 31.176, -75.803]
  Call Extruder(658.15610)
  MoveL 10634 to (233.14, 162.55, 144.49) mm, rotated rx -180 ry 0 rz 180 deg; joints [-30.426, 14.021, 68.692, 77.813, 31.205, -75.829]
  MoveL 10635 to (233.14, 162.55, 144.49) mm, rotated rx -180 ry 0 rz 180 deg; joints [-30.426, 14.021, 68.692, 77.813, 31.205, -75.829]
  Call Extruder(658.33777)
  MoveL 10636 to (232.87, 162.69, 144.49) mm, rotated rx -180 ry 0 rz 180 deg; joints [-30.453, 13.992, 68.728, 77.837, 31.23, -75.853]
  MoveL 10637 to (232.87, 162.69, 144.49) mm, rotated rx -180 ry 0 rz 180 deg; joints [-30.453, 13.992, 68.728, 77.837, 31.23, -75.853]
  Call Extruder(658.49574)
  MoveL 10638 to (232.62, 162.8, 144.49) mm, rotated rx 180 ry 0 rz 180 deg; joints [-30.476, 13.963, 68.763, 77.858, 31.25, -75.874]
  MoveL 10639 to (232.62, 162.8, 144.49) mm, rotated rx 180 ry 0 rz 180 deg; joints [-30.476, 13.963, 68.763, 77.858, 31.25, -75.874]
  Call Extruder(658.65309)
  MoveL 10640 to (232.37, 162.91, 144.49) mm, rotated rx 180 ry 0 rz -180 deg; joints [-30.498, 13.935, 68.798, 77.879, 31.271, -75.895]
  MoveL 10641 to (232.37, 162.91, 144.49) mm, rotated rx 180 ry 0 rz -180 deg; joints [-30.498, 13.935, 68.798, 77.879, 31.271, -75.895]
  Call Extruder(658.83583)
  MoveL 10642 to (232.08, 163.03, 144.49) mm, rotated rx 180 ry 0 rz 180 deg; joints [-30.524, 13.901, 68.839, 77.903, 31.295, -75.92]
  MoveL 10643 to (232.08, 163.03, 144.49) mm, rotated rx 180 ry 0 rz 180 deg; joints [-30.524, 13.901, 68.839, 77.903, 31.295, -75.92]
  Call Extruder(659.01781)
  MoveL 10644 to (231.78, 163.15, 144.49) mm, rotated rx 180 ry 0 rz 180 deg; joints [-30.551, 13.867, 68.881, 77.928, 31.318, -75.945]
  MoveL 10645 to (231.78, 163.15, 144.49) mm, rotated rx 180 ry 0 rz 180 deg; joints [-30.551, 13.867, 68.881, 77.928, 31.318, -75.945]
  Call Extruder(659.16515)
  MoveL 10646 to (231.54, 163.24, 144.49) mm, rotated rx 180 ry 0 rz -180 deg; joints [-30.571, 13.839, 68.916, 77.948, 31.337, -75.965]
  MoveL 10647 to (231.54, 163.24, 144.49) mm, rotated rx 180 ry 0 rz -180 deg; joints [-30.571, 13.839, 68.916, 77.948, 31.337, -75.965]
  Call Extruder(659.27837)
  MoveL 10648 to (231.35, 163.3, 144.49) mm, rotated rx -180 ry 0 rz 180 deg; joints [-30.587, 13.815, 68.944, 77.963, 31.351, -75.981]
  MoveL 10649 to (231.35, 163.3, 144.49) mm, rotated rx -180 ry 0 rz 180 deg; joints [-30.587, 13.815, 68.944, 77.963, 31.351, -75.981]
  Call Extruder(659.39115)
  MoveL 10650 to (231.17, 163.36, 144.49) mm, rotated rx 180 ry 0 rz 180 deg; joints [-30.602, 13.792, 68.972, 77.979, 31.365, -75.997]
  MoveL 10651 to (231.17, 163.36, 144.49) mm, rotated rx 180 ry 0 rz 180 deg; joints [-30.602, 13.792, 68.972, 77.979, 31.365, -75.997]
  Call Extruder(659.50349)
  MoveL 10652 to (230.98, 163.42, 144.49) mm, rotated rx 180 ry 0 rz -180 deg; joints [-30.618, 13.769, 69.001, 77.994, 31.379, -76.013]
  MoveL 10653 to (230.98, 163.42, 144.49) mm, rotated rx 180 ry 0 rz -180 deg; joints [-30.618, 13.769, 69.001, 77.994, 31.379, -76.013]
  Call Extruder(659.61538)
  MoveL 10654 to (230.79, 163.48, 144.49) mm, rotated rx 180 ry 0 rz 180 deg; joints [-30.633, 13.746, 69.029, 78.01, 31.393, -76.028]
  MoveL 10655 to (230.79, 163.48, 144.49) mm, rotated rx 180 ry 0 rz 180 deg; joints [-30.633, 13.746, 69.029, 78.01, 31.393, -76.028]
  Call Extruder(659.73678)
  MoveL 10656 to (230.58, 163.55, 144.49) mm, rotated rx 180 ry 0 rz 180 deg; joints [-30.65, 13.72, 69.06, 78.027, 31.408, -76.046]
  MoveL 10657 to (230.58, 163.55, 144.49) mm, rotated rx 180 ry 0 rz 180 deg; joints [-30.65, 13.72, 69.06, 78.027, 31.408, -76.046]
  Call Extruder(659.86760)
  MoveL 10658 to (230.36, 163.62, 144.49) mm, rotated rx -180 ry 0 rz -180 deg; joints [-30.668, 13.692, 69.095, 78.045, 31.424, -76.064]
  MoveL 10659 to (230.36, 163.62, 144.49) mm, rotated rx -180 ry 0 rz -180 deg; joints [-30.668, 13.692, 69.095, 78.045, 31.424, -76.064]
  Call Extruder(659.99784)
  MoveL 10660 to (230.14, 163.68, 144.49) mm, rotated rx -180 ry 0 rz 180 deg; joints [-30.685, 13.664, 69.129, 78.063, 31.44, -76.083]
  MoveL 10661 to (230.14, 163.68, 144.49) mm, rotated rx -180 ry 0 rz 180 deg; joints [-30.685, 13.664, 69.129, 78.063, 31.44, -76.083]
  Call Extruder(660.12753)
  MoveL 10662 to (229.91, 163.75, 144.49) mm, rotated rx -180 ry 0 rz -180 deg; joints [-30.703, 13.636, 69.163, 78.081, 31.456, -76.102]
  MoveL 10663 to (229.91, 163.75, 144.49) mm, rotated rx -180 ry 0 rz -180 deg; joints [-30.703, 13.636, 69.163, 78.081, 31.456, -76.102]
  Call Extruder(660.25665)
  MoveL 10664 to (229.69, 163.82, 144.49) mm, rotated rx -180 ry 0 rz 180 deg; joints [-30.721, 13.608, 69.197, 78.099, 31.472, -76.12]
  MoveL 10665 to (229.69, 163.82, 144.49) mm, rotated rx -180 ry 0 rz 180 deg; joints [-30.721, 13.608, 69.197, 78.099, 31.472, -76.12]
  Call Extruder(660.37172)
  MoveL 10666 to (229.48, 163.86, 144.49) mm, rotated rx 180 ry 0 rz 180 deg; joints [-30.736, 13.582, 69.23, 78.115, 31.485, -76.137]
  MoveL 10667 to (229.48, 163.86, 144.49) mm, rotated rx 180 ry 0 rz 180 deg; joints [-30.736, 13.582, 69.23, 78.115, 31.485, -76.137]
  Call Extruder(660.48634)
  MoveL 10668 to (229.28, 163.91, 144.49) mm, rotated rx 180 ry 0 rz 180 deg; joints [-30.751, 13.555, 69.263, 78.132, 31.499, -76.154]
  MoveL 10669 to (229.28, 163.91, 144.49) mm, rotated rx 180 ry 0 rz 180 deg; joints [-30.751, 13.555, 69.263, 78.132, 31.499, -76.154]
  Call Extruder(660.60051)
  MoveL 10670 to (229.08, 163.95, 144.49) mm, rotated rx 180 ry 0 rz -180 deg; joints [-30.766, 13.528, 69.295, 78.148, 31.512, -76.171]
  MoveL 10671 to (229.08, 163.95, 144.49) mm, rotated rx 180 ry 0 rz -180 deg; joints [-30.766, 13.528, 69.295, 78.148, 31.512, -76.171]
  Call Extruder(660.71423)
  MoveL 10672 to (228.87, 164, 144.49) mm, rotated rx -180 ry 0 rz 180 deg; joints [-30.781, 13.501, 69.328, 78.164, 31.525, -76.188]
  MoveL 10673 to (228.87, 164, 144.49) mm, rotated rx -180 ry 0 rz 180 deg; joints [-30.781, 13.501, 69.328, 78.164, 31.525, -76.188]
  Call Extruder(660.83965)
  MoveL 10674 to (228.64, 164.04, 144.49) mm, rotated rx -180 ry 0 rz 180 deg; joints [-30.797, 13.47, 69.365, 78.182, 31.539, -76.206]
  MoveL 10675 to (228.64, 164.04, 144.49) mm, rotated rx -180 ry 0 rz 180 deg; joints [-30.797, 13.47, 69.365, 78.182, 31.539, -76.206]
  Call Extruder(660.97663)
  MoveL 10676 to (228.4, 164.09, 144.49) mm, rotated rx 180 ry 0 rz 180 deg; joints [-30.815, 13.437, 69.405, 78.201, 31.555, -76.227]
  MoveL 10677 to (228.4, 164.09, 144.49) mm, rotated rx 180 ry 0 rz 180 deg; joints [-30.815, 13.437, 69.405, 78.201, 31.555, -76.227]
  Call Extruder(661.11299)
  MoveL 10678 to (228.15, 164.14, 144.49) mm, rotated rx 180 ry 0 rz 180 deg; joints [-30.832, 13.404, 69.446, 78.221, 31.571, -76.247]
  MoveL 10679 to (228.15, 164.14, 144.49) mm, rotated rx 180 ry 0 rz 180 deg; joints [-30.832, 13.404, 69.446, 78.221, 31.571, -76.247]
  Call Extruder(661.24875)
  MoveL 10680 to (227.9, 164.19, 144.49) mm, rotated rx -180 ry 0 rz 180 deg; joints [-30.85, 13.371, 69.487, 78.241, 31.587, -76.267]
  MoveL 10681 to (227.9, 164.19, 144.49) mm, rotated rx -180 ry 0 rz 180 deg; joints [-30.85, 13.371, 69.487, 78.241, 31.587, -76.267]
  Call Extruder(661.38390)
  MoveL 10682 to (227.65, 164.24, 144.49) mm, rotated rx 180 ry 0 rz 180 deg; joints [-30.868, 13.337, 69.527, 78.26, 31.602, -76.288]
  MoveL 10683 to (227.65, 164.24, 144.49) mm, rotated rx 180 ry 0 rz 180 deg; joints [-30.868, 13.337, 69.527, 78.26, 31.602, -76.288]
  Call Extruder(661.51844)
  MoveL 10684 to (227.4, 164.29, 144.49) mm, rotated rx 180 ry 0 rz 180 deg; joints [-30.886, 13.304, 69.567, 78.279, 31.618, -76.308]
  MoveL 10685 to (227.4, 164.29, 144.49) mm, rotated rx 180 ry 0 rz 180 deg; joints [-30.886, 13.304, 69.567, 78.279, 31.618, -76.308]
  Call Extruder(661.65236)
  MoveL 10686 to (227.15, 164.34, 144.49) mm, rotated rx 180 ry 0 rz -180 deg; joints [-30.903, 13.271, 69.608, 78.299, 31.634, -76.328]
  MoveL 10687 to (227.15, 164.34, 144.49) mm, rotated rx 180 ry 0 rz -180 deg; joints [-30.903, 13.271, 69.608, 78.299, 31.634, -76.328]
  Call Extruder(661.80023)
  MoveL 10688 to (226.87, 164.39, 144.49) mm, rotated rx -180 ry 0 rz -180 deg; joints [-30.923, 13.234, 69.653, 78.32, 31.651, -76.35]
  MoveL 10689 to (226.87, 164.39, 144.49) mm, rotated rx -180 ry 0 rz -180 deg; joints [-30.923, 13.234, 69.653, 78.32, 31.651, -76.35]
  Call Extruder(661.96197)
  MoveL 10690 to (226.57, 164.44, 144.49) mm, rotated rx 180 ry 0 rz 180 deg; joints [-30.943, 13.192, 69.704, 78.344, 31.669, -76.375]
  MoveL 10691 to (226.57, 164.44, 144.49) mm, rotated rx 180 ry 0 rz 180 deg; joints [-30.943, 13.192, 69.704, 78.344, 31.669, -76.375]
  Call Extruder(662.12298)
  MoveL 10692 to (226.26, 164.49, 144.49) mm, rotated rx 180 ry 0 rz 180 deg; joints [-30.964, 13.15, 69.754, 78.367, 31.688, -76.399]
  MoveL 10693 to (226.26, 164.49, 144.49) mm, rotated rx 180 ry 0 rz 180 deg; joints [-30.964, 13.15, 69.754, 78.367, 31.688, -76.399]
  Call Extruder(662.28327)
  MoveL 10694 to (225.96, 164.54, 144.49) mm, rotated rx -180 ry 0 rz 180 deg; joints [-30.985, 13.108, 69.805, 78.39, 31.706, -76.424]
  MoveL 10695 to (225.96, 164.54, 144.49) mm, rotated rx -180 ry 0 rz 180 deg; joints [-30.985, 13.108, 69.805, 78.39, 31.706, -76.424]
  Call Extruder(662.44282)
  MoveL 10696 to (225.65, 164.58, 144.49) mm, rotated rx 180 ry 0 rz -180 deg; joints [-31.006, 13.067, 69.855, 78.413, 31.725, -76.448]
  MoveL 10697 to (225.65, 164.58, 144.49) mm, rotated rx 180 ry 0 rz -180 deg; joints [-31.006, 13.067, 69.855, 78.413, 31.725, -76.448]
  Call Extruder(662.60165)
  MoveL 10698 to (225.34, 164.63, 144.49) mm, rotated rx -180 ry 0 rz 180 deg; joints [-31.027, 13.025, 69.906, 78.437, 31.743, -76.472]
  MoveL 10699 to (225.34, 164.63, 144.49) mm, rotated rx -180 ry 0 rz 180 deg; joints [-31.027, 13.025, 69.906, 78.437, 31.743, -76.472]
  Call Extruder(662.78032)
  MoveL 10700 to (225, 164.68, 144.49) mm, rotated rx 180 ry 0 rz 180 deg; joints [-31.049, 12.977, 69.964, 78.463, 31.763, -76.5]
  MoveL 10701 to (225, 164.68, 144.49) mm, rotated rx 180 ry 0 rz 180 deg; joints [-31.049, 12.977, 69.964, 78.463, 31.763, -76.5]
  Call Extruder(662.97876)
  MoveL 10702 to (224.61, 164.73, 144.49) mm, rotated rx 180 ry 0 rz -180 deg; joints [-31.074, 12.923, 70.029, 78.492, 31.786, -76.53]
  MoveL 10703 to (224.61, 164.73, 144.49) mm, rotated rx 180 ry 0 rz -180 deg; joints [-31.074, 12.923, 70.029, 78.492, 31.786, -76.53]
  Call Extruder(663.17634)
  MoveL 10704 to (224.22, 164.77, 144.49) mm, rotated rx 180 ry 0 rz -180 deg; joints [-31.1, 12.869, 70.094, 78.521, 31.808, -76.56]
  MoveL 10705 to (224.22, 164.77, 144.49) mm, rotated rx 180 ry 0 rz -180 deg; joints [-31.1, 12.869, 70.094, 78.521, 31.808, -76.56]
  Call Extruder(663.37305)
  MoveL 10706 to (223.84, 164.82, 144.49) mm, rotated rx 180 ry 0 rz 180 deg; joints [-31.125, 12.815, 70.159, 78.549, 31.83, -76.591]
  MoveL 10707 to (223.84, 164.82, 144.49) mm, rotated rx 180 ry 0 rz 180 deg; joints [-31.125, 12.815, 70.159, 78.549, 31.83, -76.591]
  Call Extruder(663.56888)
  MoveL 10708 to (223.45, 164.86, 144.49) mm, rotated rx 180 ry 0 rz 180 deg; joints [-31.15, 12.761, 70.225, 78.578, 31.852, -76.621]
  MoveL 10709 to (223.45, 164.86, 144.49) mm, rotated rx 180 ry 0 rz 180 deg; joints [-31.15, 12.761, 70.225, 78.578, 31.852, -76.621]
  Call Extruder(663.86424)
  MoveL 10710 to (222.86, 164.91, 144.49) mm, rotated rx -180 ry 0 rz 180 deg; joints [-31.186, 12.677, 70.326, 78.621, 31.884, -76.666]
  MoveL 10711 to (222.86, 164.91, 144.49) mm, rotated rx -180 ry 0 rz 180 deg; joints [-31.186, 12.677, 70.326, 78.621, 31.884, -76.666]
  Call Extruder(664.15827)
  MoveL 10712 to (222.27, 164.95, 144.49) mm, rotated rx -180 ry 0 rz -180 deg; joints [-31.222, 12.593, 70.427, 78.664, 31.916, -76.711]
  MoveL 10713 to (222.27, 164.95, 144.49) mm, rotated rx -180 ry 0 rz -180 deg; joints [-31.222, 12.593, 70.427, 78.664, 31.916, -76.711]
  Call Extruder(664.45096)
  MoveL 10714 to (221.68, 165, 144.49) mm, rotated rx 180 ry 0 rz 180 deg; joints [-31.258, 12.51, 70.527, 78.706, 31.948, -76.756]
  MoveL 10715 to (221.68, 165, 144.49) mm, rotated rx 180 ry 0 rz 180 deg; joints [-31.258, 12.51, 70.527, 78.706, 31.948, -76.756]
  Call Extruder(665.02441)
  MoveL 10716 to (220.52, 165.05, 144.49) mm, rotated rx 180 ry 0 rz 180 deg; joints [-31.326, 12.341, 70.731, 78.789, 32.007, -76.844]
  MoveL 10717 to (220.52, 165.05, 144.49) mm, rotated rx 180 ry 0 rz 180 deg; joints [-31.326, 12.341, 70.731, 78.789, 32.007, -76.844]
  Call Extruder(665.73842)
  MoveL 10718 to (219.06, 165.09, 144.49) mm, rotated rx 180 ry 0 rz 180 deg; joints [-31.409, 12.128, 70.985, 78.89, 32.08, -76.952]
  Call Extruder(782.58519)
  MoveL 10719 to (-19.06, 165.09, 144.49) mm, rotated rx 180 ry 0 rz 180 deg; joints [-51.475, -16.268, 98.431, 83.805, 51.9, -80.022]
  Call Extruder(783.01380)
  MoveL 10720 to (-19.94, 165.07, 144.49) mm, rotated rx 180 ry 0 rz 180 deg; joints [-51.582, -16.35, 98.492, 83.811, 52.007, -80.009]
  MoveL 10721 to (-19.94, 165.07, 144.49) mm, rotated rx 180 ry 0 rz 180 deg; joints [-51.582, -16.35, 98.492, 83.811, 52.007, -80.009]
  Call Extruder(783.58725)
  MoveL 10722 to (-21.1, 165.03, 144.49) mm, rotated rx -180 ry 0 rz -180 deg; joints [-51.722, -16.462, 98.574, 83.819, 52.149, -79.991]
  MoveL 10723 to (-21.1, 165.03, 144.49) mm, rotated rx -180 ry 0 rz -180 deg; joints [-51.722, -16.462, 98.574, 83.819, 52.149, -79.991]
  Call Extruder(784.02155)
  MoveL 10724 to (-21.97, 164.98, 144.49) mm, rotated rx -180 ry 0 rz 180 deg; joints [-51.827, -16.547, 98.637, 83.825, 52.255, -79.977]
  MoveL 10725 to (-21.97, 164.98, 144.49) mm, rotated rx -180 ry 0 rz 180 deg; joints [-51.827, -16.547, 98.637, 83.825, 52.255, -79.977]
  Call Extruder(784.31557)
  MoveL 10726 to (-22.56, 164.93, 144.49) mm, rotated rx -180 ry 0 rz -180 deg; joints [-51.897, -16.606, 98.68, 83.828, 52.325, -79.966]
  MoveL 10727 to (-22.56, 164.93, 144.49) mm, rotated rx -180 ry 0 rz -180 deg; joints [-51.897, -16.606, 98.68, 83.828, 52.325, -79.966]
  Call Extruder(784.61093)
  MoveL 10728 to (-23.15, 164.89, 144.49) mm, rotated rx 180 ry 0 rz -180 deg; joints [-51.966, -16.665, 98.723, 83.831, 52.395, -79.955]
  MoveL 10729 to (-23.15, 164.89, 144.49) mm, rotated rx 180 ry 0 rz -180 deg; joints [-51.966, -16.665, 98.723, 83.831, 52.395, -79.955]
  Call Extruder(784.85715)
  MoveL 10730 to (-23.64, 164.84, 144.49) mm, rotated rx 180 ry 0 rz 180 deg; joints [-52.023, -16.715, 98.759, 83.833, 52.452, -79.946]
  MoveL 10731 to (-23.64, 164.84, 144.49) mm, rotated rx 180 ry 0 rz 180 deg; joints [-52.023, -16.715, 98.759, 83.833, 52.452, -79.946]
  Call Extruder(785.05385)
  MoveL 10732 to (-24.03, 164.79, 144.49) mm, rotated rx 180 ry 0 rz 180 deg; joints [-52.067, -16.755, 98.789, 83.835, 52.497, -79.938]
  MoveL 10733 to (-24.03, 164.79, 144.49) mm, rotated rx 180 ry 0 rz 180 deg; joints [-52.067, -16.755, 98.789, 83.835, 52.497, -79.938]
  Call Extruder(785.25143)
  MoveL 10734 to (-24.42, 164.75, 144.49) mm, rotated rx -180 ry 0 rz 180 deg; joints [-52.112, -16.796, 98.818, 83.836, 52.542, -79.931]
  MoveL 10735 to (-24.42, 164.75, 144.49) mm, rotated rx -180 ry 0 rz 180 deg; joints [-52.112, -16.796, 98.818, 83.836, 52.542, -79.931]
  Call Extruder(785.44987)
  MoveL 10736 to (-24.8, 164.7, 144.49) mm, rotated rx -180 ry 0 rz -180 deg; joints [-52.156, -16.836, 98.848, 83.838, 52.587, -79.923]
  MoveL 10737 to (-24.8, 164.7, 144.49) mm, rotated rx -180 ry 0 rz -180 deg; joints [-52.156, -16.836, 98.848, 83.838, 52.587, -79.923]
  Call Extruder(785.64918)
  MoveL 10738 to (-25.19, 164.66, 144.49) mm, rotated rx 180 ry 0 rz -180 deg; joints [-52.2, -16.877, 98.877, 83.839, 52.632, -79.915]
  MoveL 10739 to (-25.19, 164.66, 144.49) mm, rotated rx 180 ry 0 rz -180 deg; joints [-52.2, -16.877, 98.877, 83.839, 52.632, -79.915]
  Call Extruder(785.80801)
  MoveL 10740 to (-25.5, 164.61, 144.49) mm, rotated rx 180 ry 0 rz 180 deg; joints [-52.235, -16.91, 98.901, 83.84, 52.666, -79.908]
  MoveL 10741 to (-25.5, 164.61, 144.49) mm, rotated rx 180 ry 0 rz 180 deg; joints [-52.235, -16.91, 98.901, 83.84, 52.666, -79.908]
  Call Extruder(785.96757)
  MoveL 10742 to (-25.8, 164.56, 144.49) mm, rotated rx -180 ry 0 rz 180 deg; joints [-52.269, -16.943, 98.925, 83.84, 52.701, -79.901]
  MoveL 10743 to (-25.8, 164.56, 144.49) mm, rotated rx -180 ry 0 rz 180 deg; joints [-52.269, -16.943, 98.925, 83.84, 52.701, -79.901]
  Call Extruder(786.12786)
  MoveL 10744 to (-26.11, 164.51, 144.49) mm, rotated rx -180 ry 0 rz 180 deg; joints [-52.303, -16.976, 98.949, 83.841, 52.735, -79.895]
  MoveL 10745 to (-26.11, 164.51, 144.49) mm, rotated rx -180 ry 0 rz 180 deg; joints [-52.303, -16.976, 98.949, 83.841, 52.735, -79.895]
  Call Extruder(786.28887)
  MoveL 10746 to (-26.41, 164.46, 144.49) mm, rotated rx 180 ry 0 rz 180 deg; joints [-52.337, -17.009, 98.973, 83.841, 52.77, -79.888]
  MoveL 10747 to (-26.41, 164.46, 144.49) mm, rotated rx 180 ry 0 rz 180 deg; joints [-52.337, -17.009, 98.973, 83.841, 52.77, -79.888]
  Call Extruder(786.45061)
  MoveL 10748 to (-26.72, 164.41, 144.49) mm, rotated rx 180 ry 0 rz 180 deg; joints [-52.371, -17.043, 98.997, 83.842, 52.804, -79.881]
  MoveL 10749 to (-26.72, 164.41, 144.49) mm, rotated rx 180 ry 0 rz 180 deg; joints [-52.371, -17.043, 98.997, 83.842, 52.804, -79.881]
  Call Extruder(786.61308)
  MoveL 10750 to (-27.03, 164.37, 144.49) mm, rotated rx 180 ry 0 rz 180 deg; joints [-52.405, -17.076, 99.021, 83.843, 52.839, -79.874]
  MoveL 10751 to (-27.03, 164.37, 144.49) mm, rotated rx 180 ry 0 rz 180 deg; joints [-52.405, -17.076, 99.021, 83.843, 52.839, -79.874]
  Call Extruder(786.74701)
  MoveL 10752 to (-27.28, 164.32, 144.49) mm, rotated rx 180 ry 0 rz 180 deg; joints [-52.432, -17.104, 99.042, 83.843, 52.866, -79.868]
  MoveL 10753 to (-27.28, 164.32, 144.49) mm, rotated rx 180 ry 0 rz 180 deg; joints [-52.432, -17.104, 99.042, 83.843, 52.866, -79.868]
  Call Extruder(786.88155)
  MoveL 10754 to (-27.52, 164.27, 144.49) mm, rotated rx 180 ry 0 rz 180 deg; joints [-52.459, -17.132, 99.062, 83.843, 52.894, -79.862]
  MoveL 10755 to (-27.52, 164.27, 144.49) mm, rotated rx 180 ry 0 rz 180 deg; joints [-52.459, -17.132, 99.062, 83.843, 52.894, -79.862]
  Call Extruder(787.01669)
  MoveL 10756 to (-27.77, 164.22, 144.49) mm, rotated rx 180 ry 0 rz 180 deg; joints [-52.486, -17.16, 99.083, 83.843, 52.921, -79.856]
  MoveL 10757 to (-27.77, 164.22, 144.49) mm, rotated rx 180 ry 0 rz 180 deg; joints [-52.486, -17.16, 99.083, 83.843, 52.921, -79.856]
  Call Extruder(787.15245)
  MoveL 10758 to (-28.02, 164.17, 144.49) mm, rotated rx 180 ry 0 rz -180 deg; joints [-52.513, -17.188, 99.103, 83.843, 52.948, -79.85]
  MoveL 10759 to (-28.02, 164.17, 144.49) mm, rotated rx 180 ry 0 rz -180 deg; joints [-52.513, -17.188, 99.103, 83.843, 52.948, -79.85]
  Call Extruder(787.28882)
  MoveL 10760 to (-28.27, 164.12, 144.49) mm, rotated rx 180 ry 0 rz 180 deg; joints [-52.54, -17.216, 99.123, 83.843, 52.976, -79.844]
  MoveL 10761 to (-28.27, 164.12, 144.49) mm, rotated rx 180 ry 0 rz 180 deg; joints [-52.54, -17.216, 99.123, 83.843, 52.976, -79.844]
  Call Extruder(787.42580)
  MoveL 10762 to (-28.52, 164.07, 144.49) mm, rotated rx -180 ry 0 rz 180 deg; joints [-52.567, -17.244, 99.143, 83.843, 53.003, -79.837]
  MoveL 10763 to (-28.52, 164.07, 144.49) mm, rotated rx -180 ry 0 rz 180 deg; joints [-52.567, -17.244, 99.143, 83.843, 53.003, -79.837]
  Call Extruder(787.56338)
  MoveL 10764 to (-28.77, 164.02, 144.49) mm, rotated rx 180 ry 0 rz -180 deg; joints [-52.594, -17.272, 99.164, 83.843, 53.031, -79.831]
  MoveL 10765 to (-28.77, 164.02, 144.49) mm, rotated rx 180 ry 0 rz -180 deg; joints [-52.594, -17.272, 99.164, 83.843, 53.031, -79.831]
  Call Extruder(787.67710)
  MoveL 10766 to (-28.97, 163.97, 144.49) mm, rotated rx 180 ry 0 rz 180 deg; joints [-52.616, -17.296, 99.18, 83.843, 53.053, -79.826]
  MoveL 10767 to (-28.97, 163.97, 144.49) mm, rotated rx 180 ry 0 rz 180 deg; joints [-52.616, -17.296, 99.18, 83.843, 53.053, -79.826]
  Call Extruder(787.79127)
  MoveL 10768 to (-29.18, 163.93, 144.49) mm, rotated rx 180 ry 0 rz 180 deg; joints [-52.638, -17.319, 99.197, 83.843, 53.075, -79.821]
  MoveL 10769 to (-29.18, 163.93, 144.49) mm, rotated rx 180 ry 0 rz 180 deg; joints [-52.638, -17.319, 99.197, 83.843, 53.075, -79.821]
  Call Extruder(787.90589)
  MoveL 10770 to (-29.38, 163.88, 144.49) mm, rotated rx 180 ry 0 rz 180 deg; joints [-52.659, -17.343, 99.214, 83.843, 53.097, -79.815]
  MoveL 10771 to (-29.38, 163.88, 144.49) mm, rotated rx 180 ry 0 rz 180 deg; joints [-52.659, -17.343, 99.214, 83.843, 53.097, -79.815]
  Call Extruder(788.02096)
  MoveL 10772 to (-29.59, 163.84, 144.49) mm, rotated rx 180 ry 0 rz 180 deg; joints [-52.681, -17.366, 99.231, 83.843, 53.12, -79.81]
  MoveL 10773 to (-29.59, 163.84, 144.49) mm, rotated rx 180 ry 0 rz 180 deg; joints [-52.681, -17.366, 99.231, 83.843, 53.12, -79.81]
  Call Extruder(788.14320)
  MoveL 10774 to (-29.8, 163.78, 144.49) mm, rotated rx 180 ry 0 rz 180 deg; joints [-52.703, -17.392, 99.25, 83.843, 53.142, -79.804]
  MoveL 10775 to (-29.8, 163.78, 144.49) mm, rotated rx 180 ry 0 rz 180 deg; joints [-52.703, -17.392, 99.25, 83.843, 53.142, -79.804]
  Call Extruder(788.27288)
  MoveL 10776 to (-30.02, 163.72, 144.49) mm, rotated rx 180 ry 0 rz 180 deg; joints [-52.726, -17.42, 99.27, 83.842, 53.165, -79.797]
  MoveL 10777 to (-30.02, 163.72, 144.49) mm, rotated rx 180 ry 0 rz 180 deg; joints [-52.726, -17.42, 99.27, 83.842, 53.165, -79.797]
  Call Extruder(788.40312)
  MoveL 10778 to (-30.25, 163.65, 144.49) mm, rotated rx 180 ry 0 rz -180 deg; joints [-52.748, -17.448, 99.29, 83.841, 53.187, -79.791]
  MoveL 10779 to (-30.25, 163.65, 144.49) mm, rotated rx 180 ry 0 rz -180 deg; joints [-52.748, -17.448, 99.29, 83.841, 53.187, -79.791]
  Call Extruder(788.53393)
  MoveL 10780 to (-30.47, 163.58, 144.49) mm, rotated rx -180 ry 0 rz 180 deg; joints [-52.77, -17.475, 99.31, 83.84, 53.21, -79.784]
  MoveL 10781 to (-30.47, 163.58, 144.49) mm, rotated rx -180 ry 0 rz 180 deg; joints [-52.77, -17.475, 99.31, 83.84, 53.21, -79.784]
  Call Extruder(788.66530)
  MoveL 10782 to (-30.7, 163.51, 144.49) mm, rotated rx 180 ry 0 rz -180 deg; joints [-52.792, -17.503, 99.33, 83.839, 53.233, -79.777]
  MoveL 10783 to (-30.7, 163.51, 144.49) mm, rotated rx 180 ry 0 rz -180 deg; joints [-52.792, -17.503, 99.33, 83.839, 53.233, -79.777]
  Call Extruder(788.77719)
  MoveL 10784 to (-30.88, 163.45, 144.49) mm, rotated rx 180 ry 0 rz 180 deg; joints [-52.81, -17.527, 99.347, 83.838, 53.252, -79.771]
  MoveL 10785 to (-30.88, 163.45, 144.49) mm, rotated rx 180 ry 0 rz 180 deg; joints [-52.81, -17.527, 99.347, 83.838, 53.252, -79.771]
  Call Extruder(788.88953)
  MoveL 10786 to (-31.07, 163.39, 144.49) mm, rotated rx 180 ry 0 rz 180 deg; joints [-52.829, -17.551, 99.364, 83.837, 53.27, -79.765]
  MoveL 10787 to (-31.07, 163.39, 144.49) mm, rotated rx 180 ry 0 rz 180 deg; joints [-52.829, -17.551, 99.364, 83.837, 53.27, -79.765]
  Call Extruder(789.00231)
  MoveL 10788 to (-31.26, 163.33, 144.49) mm, rotated rx 180 ry 0 rz 180 deg; joints [-52.847, -17.575, 99.381, 83.836, 53.289, -79.759]
  MoveL 10789 to (-31.26, 163.33, 144.49) mm, rotated rx 180 ry 0 rz 180 deg; joints [-52.847, -17.575, 99.381, 83.836, 53.289, -79.759]
  Call Extruder(789.11553)
  MoveL 10790 to (-31.45, 163.27, 144.49) mm, rotated rx 180 ry 0 rz 180 deg; joints [-52.866, -17.599, 99.398, 83.835, 53.308, -79.753]
  MoveL 10791 to (-31.45, 163.27, 144.49) mm, rotated rx 180 ry 0 rz 180 deg; joints [-52.866, -17.599, 99.398, 83.835, 53.308, -79.753]
  Call Extruder(789.22920)
  MoveL 10792 to (-31.64, 163.21, 144.49) mm, rotated rx 180 ry 0 rz 180 deg; joints [-52.884, -17.623, 99.415, 83.834, 53.327, -79.747]
  MoveL 10793 to (-31.64, 163.21, 144.49) mm, rotated rx 180 ry 0 rz 180 deg; joints [-52.884, -17.623, 99.415, 83.834, 53.327, -79.747]
  Call Extruder(789.41118)
  MoveL 10794 to (-31.93, 163.09, 144.49) mm, rotated rx 180 ry 0 rz 180 deg; joints [-52.91, -17.663, 99.444, 83.831, 53.354, -79.736]
  MoveL 10795 to (-31.93, 163.09, 144.49) mm, rotated rx 180 ry 0 rz 180 deg; joints [-52.91, -17.663, 99.444, 83.831, 53.354, -79.736]
  Call Extruder(789.59392)
  MoveL 10796 to (-32.22, 162.97, 144.49) mm, rotated rx 180 ry 0 rz -180 deg; joints [-52.936, -17.703, 99.472, 83.829, 53.381, -79.726]
  MoveL 10797 to (-32.22, 162.97, 144.49) mm, rotated rx 180 ry 0 rz -180 deg; joints [-52.936, -17.703, 99.472, 83.829, 53.381, -79.726]
  Call Extruder(789.76433)
  MoveL 10798 to (-32.49, 162.85, 144.49) mm, rotated rx -180 ry 0 rz 180 deg; joints [-52.96, -17.74, 99.499, 83.826, 53.405, -79.716]
  MoveL 10799 to (-32.49, 162.85, 144.49) mm, rotated rx -180 ry 0 rz 180 deg; joints [-52.96, -17.74, 99.499, 83.826, 53.405, -79.716]
  Call Extruder(789.92231)
  MoveL 10800 to (-32.74, 162.74, 144.49) mm, rotated rx 180 ry 0 rz 180 deg; joints [-52.982, -17.775, 99.524, 83.824, 53.428, -79.706]
  MoveL 10801 to (-32.74, 162.74, 144.49) mm, rotated rx 180 ry 0 rz 180 deg; joints [-52.982, -17.775, 99.524, 83.824, 53.428, -79.706]
  Call Extruder(790.08088)
  MoveL 10802 to (-32.99, 162.64, 144.49) mm, rotated rx 180 ry 0 rz -180 deg; joints [-53.004, -17.809, 99.548, 83.821, 53.451, -79.697]
  MoveL 10803 to (-32.99, 162.64, 144.49) mm, rotated rx 180 ry 0 rz -180 deg; joints [-53.004, -17.809, 99.548, 83.821, 53.451, -79.697]
  Call Extruder(790.28705)
  MoveL 10804 to (-33.29, 162.46, 144.49) mm, rotated rx 180 ry 0 rz 180 deg; joints [-53.026, -17.857, 99.582, 83.816, 53.474, -79.683]
  MoveL 10805 to (-33.29, 162.46, 144.49) mm, rotated rx 180 ry 0 rz 180 deg; joints [-53.026, -17.857, 99.582, 83.816, 53.474, -79.683]
  Call Extruder(790.49399)
  MoveL 10806 to (-33.6, 162.29, 144.49) mm, rotated rx 180 ry 0 rz -180 deg; joints [-53.049, -17.904, 99.616, 83.811, 53.498, -79.669]
  MoveL 10807 to (-33.6, 162.29, 144.49) mm, rotated rx 180 ry 0 rz -180 deg; joints [-53.049, -17.904, 99.616, 83.811, 53.498, -79.669]
  Call Extruder(790.70172)
  MoveL 10808 to (-33.9, 162.11, 144.49) mm, rotated rx 180 ry 0 rz -180 deg; joints [-53.071, -17.952, 99.65, 83.806, 53.521, -79.655]
  MoveL 10809 to (-33.9, 162.11, 144.49) mm, rotated rx 180 ry 0 rz -180 deg; joints [-53.071, -17.952, 99.65, 83.806, 53.521, -79.655]
  Call Extruder(790.91022)
  MoveL 10810 to (-34.21, 161.93, 144.49) mm, rotated rx 180 ry 0 rz 180 deg; joints [-53.094, -17.999, 99.683, 83.801, 53.545, -79.641]
  MoveL 10811 to (-34.21, 161.93, 144.49) mm, rotated rx 180 ry 0 rz 180 deg; joints [-53.094, -17.999, 99.683, 83.801, 53.545, -79.641]
  Call Extruder(791.08976)
  MoveL 10812 to (-34.45, 161.76, 144.49) mm, rotated rx -180 ry 0 rz 180 deg; joints [-53.109, -18.042, 99.713, 83.795, 53.561, -79.628]
  MoveL 10813 to (-34.45, 161.76, 144.49) mm, rotated rx -180 ry 0 rz 180 deg; joints [-53.109, -18.042, 99.713, 83.795, 53.561, -79.628]
  Call Extruder(791.42319)
  MoveL 10814 to (-34.9, 161.43, 144.49) mm, rotated rx -180 ry 0 rz 180 deg; joints [-53.135, -18.12, 99.769, 83.784, 53.59, -79.603]
  MoveL 10815 to (-34.9, 161.43, 144.49) mm, rotated rx -180 ry 0 rz 180 deg; joints [-53.135, -18.12, 99.769, 83.784, 53.59, -79.603]
  Call Extruder(791.75781)
  MoveL 10816 to (-35.35, 161.1, 144.49) mm, rotated rx 180 ry 0 rz 180 deg; joints [-53.163, -18.198, 99.824, 83.774, 53.619, -79.578]
  Call Extruder(792.58572)
  MoveL 10817 to (-36.39, 160.19, 144.49) mm, rotated rx 180 ry 0 rz 180 deg; joints [-53.209, -18.397, 99.964, 83.741, 53.671, -79.512]
  Call Extruder(793.10708)
  MoveL 10818 to (-36.97, 159.54, 144.49) mm, rotated rx -180 ry 0 rz 180 deg; joints [-53.221, -18.524, 100.053, 83.716, 53.687, -79.467]
  Set speed (130.0 mm/s)
  MoveL 10819 to (-38.97, 156.79, 144.49) mm, rotated rx -180 ry 0 rz 180 deg; joints [-53.214, -19.023, 100.401, 83.604, 53.697, -79.279]
